// TIA Portal V20 export
FUNCTION_BLOCK "CallEquipment"   // FB29, LAD
TITLE = CallEquipment
AUTHOR : ERsystem_FA2_DH. Kim
// This block contains the logic and futher calls (e.g. sequences, control modules, diagnostics etc.) of the equipment module.
// stored: IsIECCheckEnabled true, MemoryReserve 100, Namespace Unit1.Em5, SetENOAutomatically false
   VAR_INPUT
      ZoneOperationEnable { ExternalWritable := 'False'} : "LWONIK_typeSafetyZoneManualOperation";
   END_VAR
   VAR_IN_OUT
      unitStatus : "LAF_typeUnitStatus";   // Current unit status o be used in this EM
      unitAlarmDB : "LAF_typeAlarms";   // Summarized EM Alarms for the Unit
      emFeedback : "LUC_typeEmFeedback";   // Feedback of the EM to the Unit
   END_VAR
   VAR
      InstSequenceMainPnP { S7_SetPoint := 'True'} : "Unit1.Em5.Sequence_1_MainPnP";   // EM Sequence Instance
      InstSequenceAlignTable { S7_SetPoint := 'True'} : "Unit1.Em5.Sequence_2_AlignTable";
      InstSequenceNgPnP { S7_SetPoint := 'True'} : "Unit1.Em5.Sequence_3_NgPnP";
      InstSequenceGaugeRnR : "Unit1.Em5.Sequence_10_GaugeRnR";
      instMainPnPHomeJob10 : "LAF_SelectJob";
      instMainPnPHomeJob1 : "LAF_SelectJob";
      instMainPnPLoadJob2 : "LAF_SelectJob";
      instMainPnPUnloadJob3 : "LAF_SelectJob";
      instMainPnPAvoidJob4 : "LAF_SelectJob";
      instMainPnPOneLoadJob5 : "LAF_SelectJob";
      instMainPnPOneUnLoadJob6 : "LAF_SelectJob";
      instAlignTableHomeJob1 : "LAF_SelectJob";
      instAlignTableLoadJob2 : "LAF_SelectJob";
      instAlignTableVisionJob3 : "LAF_SelectJob";
      instAlignTableUnloadJob4 : "LAF_SelectJob";
      instAlignTableMotionJob22 : "LAF_SelectJob";
      instNgPnPHomeJob1 : "LAF_SelectJob";
      instNgPnPLoadJob2 : "LAF_SelectJob";
      instNgPnPUnloadJob3 : "LAF_SelectJob";
      instGaugeRnRCommonReadyJob1 : "LAF_SelectJob";
      instGaugeRnRCommonGetMasterPieceJob2 : "LAF_SelectJob";
      instGaugeRnRCommonMainPnPMoveAlignTableStackTableJob3 : "LAF_SelectJob";
      instGaugeRnRCommonMainPnp1ToAlignTableJob4 : "LAF_SelectJob";
      instGaugeRnRCommonMainPnPMoveReelCutConvyorAlignTableJob5 : "LAF_SelectJob";
      instGaugeRnRCommonAlignTableVisionAdjustJob6 : "LAF_SelectJob";
      instGaugeRnR1AlignAlignTableToMainPnP1Job10 { S7_SetPoint := 'True'} : "LAF_SelectJob";
      instGaugeRnR1AlignMainPnPMoveReelCutConvyorAlignTableJob11 { S7_SetPoint := 'True'} : "LAF_SelectJob";
      instGaugeRnR1AlignAlignTableMoveWaitJob12 { S7_SetPoint := 'True'} : "LAF_SelectJob";
      instGaugeRnR1AlignUnloadMasterPieceJob13 { S7_SetPoint := 'True'} : "LAF_SelectJob";
      instGaugeRnR1StackMainPnPMoveReelCutConvyorAlignTableJob15 { S7_SetPoint := 'True'} : "LAF_SelectJob";
      instGaugeRnR1StackAlignTableToMainPnP2Job16 { S7_SetPoint := 'True'} : "LAF_SelectJob";
      instGaugeRnR1StackMainPnPMoveAlignTableJob17 { S7_SetPoint := 'True'} : "LAF_SelectJob";
      instGaugeRnR1StackAlignTableMoveWaitJob18 { S7_SetPoint := 'True'} : "LAF_SelectJob";
      instGaugeRnR1StackMainPnP2ToStackTableJob19 { S7_SetPoint := 'True'} : "LAF_SelectJob";
      instGaugeRnR1StackStackTableToMainPnP2Job20 { S7_SetPoint := 'True'} : "LAF_SelectJob";
      instGaugeRnR1StackMainPnPMoveReelCutConvyorAlignTableJob21 { S7_SetPoint := 'True'} : "LAF_SelectJob";
      instGaugeRnR1StackMainPnP2ToAlignTableJob22 { S7_SetPoint := 'True'} : "LAF_SelectJob";
      instGaugeRnR1StackMainPnPMoveAlignTableJob23 { S7_SetPoint := 'True'} : "LAF_SelectJob";
      instGaugeRnR1StackAlignTableToMainPnP1Job24 { S7_SetPoint := 'True'} : "LAF_SelectJob";
      instGaugeRnR1StackMainPnPMoveReelCutConvyorAlignTableJob25 { S7_SetPoint := 'True'} : "LAF_SelectJob";
      instGaugeRnR1StackUnloadMasterPieceJob26 { S7_SetPoint := 'True'} : "LAF_SelectJob";
      instGaugeRnR3AlignMainPnPMoveReelCutConvyorAlignTableJob30 { S7_SetPoint := 'True'} : "LAF_SelectJob";
      instGaugeRnR3AlignNGPnPLoadMasterPieceJob31 { S7_SetPoint := 'True'} : "LAF_SelectJob";
      instGaugeRnR3AlignMainPnP2MoveAlignTableJob32 { S7_SetPoint := 'True'} : "LAF_SelectJob";
      instGaugeRnR3AlignAlignTableMoveWaitJob33 { S7_SetPoint := 'True'} : "LAF_SelectJob";
      instGaugeRnRCommonCheckCompleteJob39 { S7_SetPoint := 'True'} : "LAF_SelectJob";
      instCmPnp1stCathodeDetectSensor { S7_SetPoint := 'True'} : "LBC_DigitalSignalCn";
      instCmPnp2ndCathodeDetectSensor { S7_SetPoint := 'True'} : "LBC_DigitalSignalCn";
      instCmCathodeAlignTableElectrodeDetectSensor { S7_SetPoint := 'True'} : "LBC_DigitalSignalCn";
      instCmCathodeNgBoxFullSensorDetectSensor { S7_SetPoint := 'True'} : "LBC_DigitalSignalCn";
      instCmCathodeNgBoxDetectSensor { S7_SetPoint := 'True'} : "LBC_DigitalSignalCn";
      instCmCathodeMainPnP1AxisX { S7_SetPoint := 'True'} : "LBC_Axis64Pos_TecPlcCn";
      instCmCathodeMainPnP2AxisX { S7_SetPoint := 'True'} : "LBC_Axis64Pos_TecPlcCn";
      instCmCathodeMainPnP1AxisY { S7_SetPoint := 'True'} : "LBC_Axis64Pos_TecPlcCn";
      instCmCathodeMainPnP1AxisZ { S7_SetPoint := 'True'} : "LBC_Axis64Pos_TecPlcCn";
      instCmCathodeMainPnP2AxisZ { S7_SetPoint := 'True'} : "LBC_Axis64Pos_TecPlcCn";
      instCmCathodeAlignTableAxisX { S7_SetPoint := 'True'} : "LBC_Axis64Pos_TecPlcCn";
      instCmCathodeAlignTableAxisY1 { S7_SetPoint := 'True'} : "LBC_Axis64Pos_TecPlcCn";
      instCmCathodeAlignTableAxisY2 { S7_SetPoint := 'True'} : "LBC_Axis64Pos_TecPlcCn";
      instInterlockCathodeMainPnP1AxisX { S7_SetPoint := 'True'} : "LER_Axis64Pos_InterlockSummary";
      instInterlockCathodeMainPnP1AxisY { S7_SetPoint := 'True'} : "LER_Axis64Pos_InterlockSummary";
      instInterlockCathodeMainPnP1AxisZ { S7_SetPoint := 'True'} : "LER_Axis64Pos_InterlockSummary";
      instInterlockCathodeMainPnP2AxisX { S7_SetPoint := 'True'} : "LER_Axis64Pos_InterlockSummary";
      instInterlockCathodeMainPnP2AxisZ { S7_SetPoint := 'True'} : "LER_Axis64Pos_InterlockSummary";
      instInterlockCathodeAlignTableAxisX { S7_SetPoint := 'True'} : "LER_Axis64Pos_InterlockSummary";
      instInterlockCathodeAlignTableAxisY1 { S7_SetPoint := 'True'} : "LER_Axis64Pos_InterlockSummary";
      instInterlockCathodeAlignTableAxisY2 { S7_SetPoint := 'True'} : "LER_Axis64Pos_InterlockSummary";
      instCathodeMainPnP1AxisXSoftCam : "LER_SoftCam_Interface";
      instCathodeMainPnP2AxisXSoftCam { S7_SetPoint := 'True'} : "LER_SoftCam_Interface";
      instCathodeMainPnP1AxisYSoftCam { S7_SetPoint := 'True'} : "LER_SoftCam_Interface";
      instCathodeMainPnP1AxisZSoftCam { S7_SetPoint := 'True'} : "LER_SoftCam_Interface";
      instCathodeMainPnP2AxisZSoftCam { S7_SetPoint := 'True'} : "LER_SoftCam_Interface";
      instCathodeAlignTableAxisXSoftCam { S7_SetPoint := 'True'} : "LER_SoftCam_Interface";
      instCathodeAlignTableAxisY1SoftCam { S7_SetPoint := 'True'} : "LER_SoftCam_Interface";
      instCathodeAlignTableAxisY2SoftCam { S7_SetPoint := 'True'} : "LER_SoftCam_Interface";
      instCmCathodeMainPnP1RotaryCwCcw { ExternalAccessible := 'False'; ExternalVisible := 'False'; ExternalWritable := 'False'} : "LBC_TwoWayActuatorCn";
      instCmCathodeMainPnP1stSuctionPlateVacuum { ExternalAccessible := 'False'; ExternalVisible := 'False'; ExternalWritable := 'False'} : "LBC_TwoWayActuatorCn";
      instCmCathodeMainPnP2ndSuctionPlateVacuum { ExternalAccessible := 'False'; ExternalVisible := 'False'; ExternalWritable := 'False'} : "LBC_TwoWayActuatorCn";
      instCmCathodeAlignTableSuctionPlateVacuum { ExternalAccessible := 'False'; ExternalVisible := 'False'; ExternalWritable := 'False'; S7_SetPoint := 'True'} : "LBC_TwoWayActuatorCn";
      instCmCathodeGlassCleaning { ExternalAccessible := 'False'; ExternalVisible := 'False'; ExternalWritable := 'False'; S7_SetPoint := 'True'} : "LBC_TwoWayActuatorCn";
      instCmCathodeNgPnpUpDown { ExternalAccessible := 'False'; ExternalVisible := 'False'; ExternalWritable := 'False'; S7_SetPoint := 'True'} : "LBC_TwoWayActuatorCn";
      instCmCathodeNgPnp1stFwdBwd { ExternalAccessible := 'False'; ExternalVisible := 'False'; ExternalWritable := 'False'; S7_SetPoint := 'True'} : "LBC_TwoWayActuatorCn";
      instCmCathodeNgPnp2ndFwdBwd { ExternalAccessible := 'False'; ExternalVisible := 'False'; ExternalWritable := 'False'; S7_SetPoint := 'True'} : "LBC_TwoWayActuatorCn";
      instCmCathodeMaintenanceMovingFixFwdBwd { ExternalAccessible := 'False'; ExternalVisible := 'False'; ExternalWritable := 'False'; S7_SetPoint := 'True'} : "LBC_TwoWayActuatorCn";
      instCmCathodeNgBoxLiftUpDown { ExternalAccessible := 'False'; ExternalVisible := 'False'; ExternalWritable := 'False'; S7_SetPoint := 'True'} : "LBC_TwoWayActuatorCn";
      instCmCathodeNgBoxLockUpDown { ExternalAccessible := 'False'; ExternalVisible := 'False'; ExternalWritable := 'False'; S7_SetPoint := 'True'} : "LBC_TwoWayActuatorCn";
      instCmCathodeNgPnpVaccum { ExternalAccessible := 'False'; ExternalVisible := 'False'; ExternalWritable := 'False'; S7_SetPoint := 'True'} : "LBC_TwoWayActuatorCn";
      instCmCathodeConveyorCoverFwdBwd { S7_SetPoint := 'True'} : "LBC_TwoWayActuatorCn";
      instCmCathodeConveyorPickUpBlower { S7_SetPoint := 'True'} : "LBC_TwoWayActuatorCn";
      instCmCathodeVisionControllerInterface { ExternalAccessible := 'False'; ExternalVisible := 'False'; ExternalWritable := 'False'; S7_SetPoint := 'True'} : "LER_Vision_XGX2000";
      instAlignVisionConversion : "LER_AlignVisionConversion";
      instManageAlarms { ExternalWritable := 'False'} : "LAF_ManageAlarms";
      instEventsPFE : "Unit1.Em5.EventsPFE";
      instLER_BrakeTestCathodeMainPnP1AxisZ : "LER_BrakeTest";
      instLER_BrakeTestCathodeMainPnP2AxisZ { S7_SetPoint := 'True'} : "LER_BrakeTest";
      statUnitStatus { ExternalWritable := 'False'} : "LAF_typeUnitStatus";   // Unit Status used in this EM
      statSlmStatus : Struct
         running { ExternalWritable := 'False'} : Bool;
         powerOff { ExternalWritable := 'False'} : Bool;
      END_STRUCT;
      statAllBrakeTest { ExternalWritable := 'False'} : "LER_typeBrakeTestUnitCommands";
      statTonTime { ExternalAccessible := 'False'; ExternalVisible := 'False'; ExternalWritable := 'False'} : Array[0..1999] of TON_TIME;
      statTofTime { ExternalAccessible := 'False'; ExternalVisible := 'False'; ExternalWritable := 'False'} : Array[0..99] of TOF_TIME;
      statPulse { ExternalAccessible := 'False'; ExternalVisible := 'False'; ExternalWritable := 'False'} : Struct
         miscellaneous : Array[0..99] of Bool;
         workingDone : Struct
            mainPnP : Array[0..99] of Bool;
            alignTable : Array[0..99] of Bool;
            ngPnP : Array[0..99] of Bool;
         END_STRUCT;
         axisEnable : Array[0..99] of Bool;
         brakeTest : Array[0..99] of Bool;
      END_STRUCT;
      statEnableManualCmds : Bool;
      Scan_on : Bool;
      "*** Interlock Axis ***" { ExternalAccessible := 'False'; ExternalVisible := 'False'; ExternalWritable := 'False'} : Bool;
      "cathodeMainPnP1AxisX Home" { S7_SetPoint := 'True'} : "Homing.LER_Axis";
      "cathodeMainPnP1AxisX Jog_CW" { S7_SetPoint := 'True'} : "Jog.LER_Axis";
      "cathodeMainPnP1AxisX Jog_CCW" { S7_SetPoint := 'True'} : "Jog.LER_Axis";
      "cathodeMainPnP1AxisX Position_" { S7_SetPoint := 'True'} : Array[0..5] of "Position.LER_Axis";
      "cathodeMainPnP2AxisX Home" { S7_SetPoint := 'True'} : "Homing.LER_Axis";
      "cathodeMainPnP2AxisX Jog_CW" { S7_SetPoint := 'True'} : "Jog.LER_Axis";
      "cathodeMainPnP2AxisX Jog_CCW" { S7_SetPoint := 'True'} : "Jog.LER_Axis";
      "cathodeMainPnP2AxisX Position_" { S7_SetPoint := 'True'} : Array[0..5] of "Position.LER_Axis";
      "cathodeMainPnP1AxisY Home" { S7_SetPoint := 'True'} : "Homing.LER_Axis";
      "cathodeMainPnP1AxisY Jog_CW" { S7_SetPoint := 'True'} : "Jog.LER_Axis";
      "cathodeMainPnP1AxisY Jog_CCW" { S7_SetPoint := 'True'} : "Jog.LER_Axis";
      "cathodeMainPnP1AxisY Position_" { S7_SetPoint := 'True'} : Array[0..5] of "Position.LER_Axis";
      "cathodeMainPnP1AxisZ Home" { S7_SetPoint := 'True'} : "Homing.LER_Axis";
      "cathodeMainPnP1AxisZ Jog_CW" { S7_SetPoint := 'True'} : "Jog.LER_Axis";
      "cathodeMainPnP1AxisZ Jog_CCW" { S7_SetPoint := 'True'} : "Jog.LER_Axis";
      "cathodeMainPnP1AxisZ Position_" { S7_SetPoint := 'True'} : Array[0..5] of "Position.LER_Axis";
      "cathodeMainPnP2AxisZ Home" { S7_SetPoint := 'True'} : "Homing.LER_Axis";
      "cathodeMainPnP2AxisZ Jog_CW" { S7_SetPoint := 'True'} : "Jog.LER_Axis";
      "cathodeMainPnP2AxisZ Jog_CCW" { S7_SetPoint := 'True'} : "Jog.LER_Axis";
      "cathodeMainPnP2AxisZ Position_" { S7_SetPoint := 'True'} : Array[0..5] of "Position.LER_Axis";
      "cathodeAlignTableAxisX Home" { S7_SetPoint := 'True'} : "Homing.LER_Axis";
      "cathodeAlignTableAxisX Jog_CW" { S7_SetPoint := 'True'} : "Jog.LER_Axis";
      "cathodeAlignTableAxisX Jog_CCW" { S7_SetPoint := 'True'} : "Jog.LER_Axis";
      "cathodeAlignTableAxisX Position_" { S7_SetPoint := 'True'} : Array[0..5] of "Position.LER_Axis";
      "cathodeAlignTableAxisY1 Home" { S7_SetPoint := 'True'} : "Homing.LER_Axis";
      "cathodeAlignTableAxisY1 Jog_CW" { S7_SetPoint := 'True'} : "Jog.LER_Axis";
      "cathodeAlignTableAxisY1 Jog_CCW" { S7_SetPoint := 'True'} : "Jog.LER_Axis";
      "cathodeAlignTableAxisY1 Position_" { S7_SetPoint := 'True'} : Array[0..5] of "Position.LER_Axis";
      "cathodeAlignTableAxisY2 Home" { S7_SetPoint := 'True'} : "Homing.LER_Axis";
      "cathodeAlignTableAxisY2 Jog_CW" { S7_SetPoint := 'True'} : "Jog.LER_Axis";
      "cathodeAlignTableAxisY2 Jog_CCW" { S7_SetPoint := 'True'} : "Jog.LER_Axis";
      "cathodeAlignTableAxisY2 Position_" { S7_SetPoint := 'True'} : Array[0..5] of "Position.LER_Axis";
      "*** Interlock Actuator ******" { ExternalAccessible := 'False'; ExternalVisible := 'False'; ExternalWritable := 'False'} : Bool;
      "cathodeNgBoxLiftUpDown Home" { S7_SetPoint := 'True'} : "Cylinder.LER_Actuator";
      "cathodeNgBoxLiftUpDown Work" { S7_SetPoint := 'True'} : "Cylinder.LER_Actuator";
      "cathodeNgBoxLockUpDown Home" { S7_SetPoint := 'True'} : "Cylinder.LER_Actuator";
      "cathodeNgBoxLockUpDown Work" { S7_SetPoint := 'True'} : "Cylinder.LER_Actuator";
      "cathodeMaintenanceMovingFixFrontFwdBwd Home" { S7_SetPoint := 'True'} : "Cylinder.LER_Actuator";
      "cathodeMaintenanceMovingFixFrontFwdBwd Work" { S7_SetPoint := 'True'} : "Cylinder.LER_Actuator";
      "cathodeGlassCleaning Home" { S7_SetPoint := 'True'} : "Cylinder.LER_Actuator";
      "cathodeGlassCleaning Work" { S7_SetPoint := 'True'} : "Cylinder.LER_Actuator";
      "cathodeNgPnp1stFwdBwd Home" { S7_SetPoint := 'True'} : "Cylinder.LER_Actuator";
      "cathodeNgPnp1stFwdBwd Work" { S7_SetPoint := 'True'} : "Cylinder.LER_Actuator";
      "cathodeNgPnpUpDown Home" { S7_SetPoint := 'True'} : "Cylinder.LER_Actuator";
      "cathodeNgPnpUpDown Work" { S7_SetPoint := 'True'} : "Cylinder.LER_Actuator";
      "cathodeMainPnP1RotaryCwCcw Home" { S7_SetPoint := 'True'} : "Cylinder.LER_Actuator";
      "cathodeMainPnP1RotaryCwCcw Work" { S7_SetPoint := 'True'} : "Cylinder.LER_Actuator";
      "cathodeNgPnp2ndFwdBwd Home" { S7_SetPoint := 'True'} : "Cylinder.LER_Actuator";
      "cathodeNgPnp2ndFwdBwd Work" { S7_SetPoint := 'True'} : "Cylinder.LER_Actuator";
      Tracking_05 { S7_SetPoint := 'True'} : "Unit1.Em5.PartData";
      AXIS7 : "LER_CM_Name";
      AXIS13 : "LER_CM_Name";
      AXIS18 : "LER_CM_Name";
      Cylinder23 : "LER_CM_Name";
      Cylinder28 : "LER_CM_Name";
      Vaccum15 : "LER_CM_Name";
      instAlignVisionHistory { S7_SetPoint := 'True'} : "LER_visionHistory";
      instAlignMoveCalibration { S7_SetPoint := 'True'} : "LER_AlignMoveCalibration";
      instAlignThetaCalibration { S7_SetPoint := 'True'} : "LER_AlignThetaCalibration";
      instAlignSyncMove { S7_SetPoint := 'True'} : "LER_AlignSyncMove";
      citi_Ptrig : Array[0..20] of Bool;
      citiTon : Array[0..20] of TON_TIME;
      citi : Time;
      citiTest : Array[0..20] of Bool;
   END_VAR
   VAR_TEMP
      tempIndex : Int;
      tempScInProduction : Bool;   // Mode Production and StateComplete
      tempScNoProduction : Bool;   // Mode Manual and StateComplete
   END_VAR
   VAR CONSTANT
      delayTime : Time := T#3s;
      TRUE : Bool := TRUE;
      FALSE : Bool := FALSE;
      NO_JOB : DInt;   // No job
      MIN_POSITION_NUMBER : SInt;
      INIT_POSITION_NUMBER : SInt := -1;
   END_VAR
   // // statPulse.brakeTest[0] : Unit Mode Production Rising Edge
   // // statPulse.brakeTest[1] : Unit Mode Production Rising Edge Old
   // // statPulse.brakeTest[10] : Cathode Main PnP 1 Z Axis Error Pulse
   // // statPulse.brakeTest[11] : Cathode Main PnP 2 Z Axis Error Pulse
   VAR_TEMP   // added for the SCL form of the ladder/FBD networks
      _w1 : Bool;
      _w2 : Bool;
      _w3 : Bool;
      _w4 : Bool;
      _w5 : Bool;
      _w6 : Bool;
      _w7 : Bool;
      _w8 : Bool;
      _w9 : Bool;
      _w10 : Bool;
      _w11 : Bool;
   END_VAR
BEGIN

REGION Network 1: BLOCK INFO HEADER
   // (company) / (C) Copyright (year)
   // ---------------------------------------------------------------------------------
   // Title:                             (Title of this block)
   // Comment/Function: (that is implemented in the block)
   // Library/Family:           (that the source is dedicated to)
   // Author:                        (department / person in charge / contact)
   // Target System:          (test system with FW version)
   // Engineering:              TIA Portal (SW version)
   // Restrictions:               (OB types, etc.)
   // Requirements:           (hardware, technological package, etc.)
   // ---------------------------------------------------------------------------------
   // Change log table:
   // Version          | Date             | Signature      | Expert in charge  | Changes applied ------------------------|----------------------|-------------------------|--------------------------------|-----------------------
   // 001.000.000 | yyyy-mm-dd | 0x00000000 | (name of expert) | First released version
END_REGION

REGION Network 2: DESCRIPTION
   // This is a template block provided by the Automation Framework. It can be used to create an own project.
   // The Block Info Header is prepared to put in your own data.
   // Description of the block could be added here and the docu created by Code2Docu.
END_REGION

REGION Network 3: ******************** Unit Input ********************
END_REGION

REGION Network 4: Em6 Relations SoftCam
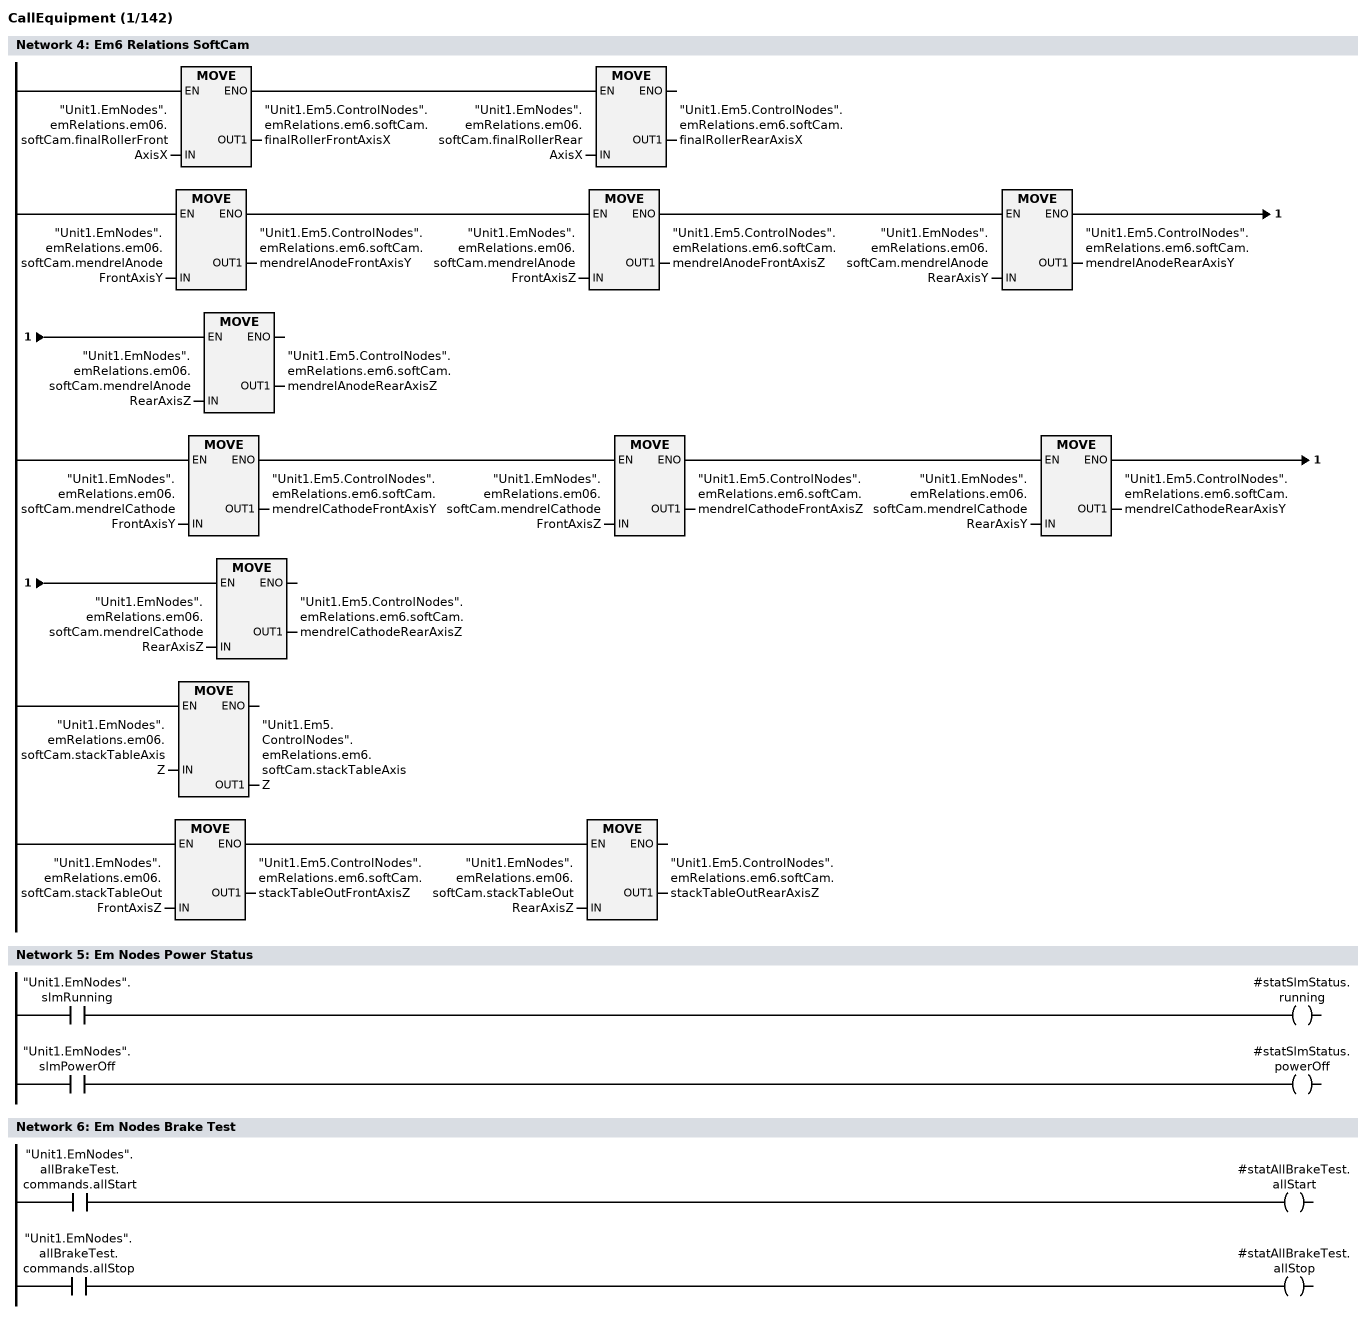
   RUNG wire#powerrail
      Move(in := "Unit1.EmNodes".emRelations.em06.softCam.finalRollerFrontAxisX, out1 => "Unit1.Em5.ControlNodes".emRelations.em6.softCam.finalRollerFrontAxisX)
      Move(in := "Unit1.EmNodes".emRelations.em06.softCam.finalRollerRearAxisX, out1 => "Unit1.Em5.ControlNodes".emRelations.em6.softCam.finalRollerRearAxisX)
   END_RUNG
   RUNG wire#powerrail
      Move(in := "Unit1.EmNodes".emRelations.em06.softCam.mendrelAnodeFrontAxisY, out1 => "Unit1.Em5.ControlNodes".emRelations.em6.softCam.mendrelAnodeFrontAxisY)
      Move(in := "Unit1.EmNodes".emRelations.em06.softCam.mendrelAnodeFrontAxisZ, out1 => "Unit1.Em5.ControlNodes".emRelations.em6.softCam.mendrelAnodeFrontAxisZ)
      Move(in := "Unit1.EmNodes".emRelations.em06.softCam.mendrelAnodeRearAxisY, out1 => "Unit1.Em5.ControlNodes".emRelations.em6.softCam.mendrelAnodeRearAxisY)
      Move(in := "Unit1.EmNodes".emRelations.em06.softCam.mendrelAnodeRearAxisZ, out1 => "Unit1.Em5.ControlNodes".emRelations.em6.softCam.mendrelAnodeRearAxisZ)
   END_RUNG
   RUNG wire#powerrail
      Move(in := "Unit1.EmNodes".emRelations.em06.softCam.mendrelCathodeFrontAxisY, out1 => "Unit1.Em5.ControlNodes".emRelations.em6.softCam.mendrelCathodeFrontAxisY)
      Move(in := "Unit1.EmNodes".emRelations.em06.softCam.mendrelCathodeFrontAxisZ, out1 => "Unit1.Em5.ControlNodes".emRelations.em6.softCam.mendrelCathodeFrontAxisZ)
      Move(in := "Unit1.EmNodes".emRelations.em06.softCam.mendrelCathodeRearAxisY, out1 => "Unit1.Em5.ControlNodes".emRelations.em6.softCam.mendrelCathodeRearAxisY)
      Move(in := "Unit1.EmNodes".emRelations.em06.softCam.mendrelCathodeRearAxisZ, out1 => "Unit1.Em5.ControlNodes".emRelations.em6.softCam.mendrelCathodeRearAxisZ)
   END_RUNG
   RUNG wire#powerrail
      Move(in := "Unit1.EmNodes".emRelations.em06.softCam.stackTableAxisZ, out1 => "Unit1.Em5.ControlNodes".emRelations.em6.softCam.stackTableAxisZ)
   END_RUNG
   RUNG wire#powerrail
      Move(in := "Unit1.EmNodes".emRelations.em06.softCam.stackTableOutFrontAxisZ, out1 => "Unit1.Em5.ControlNodes".emRelations.em6.softCam.stackTableOutFrontAxisZ)
      Move(in := "Unit1.EmNodes".emRelations.em06.softCam.stackTableOutRearAxisZ, out1 => "Unit1.Em5.ControlNodes".emRelations.em6.softCam.stackTableOutRearAxisZ)
   END_RUNG
   // the same network as SCL:
   "Unit1.Em5.ControlNodes".emRelations.em6.softCam.finalRollerFrontAxisX := "Unit1.EmNodes".emRelations.em06.softCam.finalRollerFrontAxisX;
   "Unit1.Em5.ControlNodes".emRelations.em6.softCam.finalRollerRearAxisX := "Unit1.EmNodes".emRelations.em06.softCam.finalRollerRearAxisX;
   "Unit1.Em5.ControlNodes".emRelations.em6.softCam.mendrelAnodeFrontAxisY := "Unit1.EmNodes".emRelations.em06.softCam.mendrelAnodeFrontAxisY;
   "Unit1.Em5.ControlNodes".emRelations.em6.softCam.mendrelAnodeFrontAxisZ := "Unit1.EmNodes".emRelations.em06.softCam.mendrelAnodeFrontAxisZ;
   "Unit1.Em5.ControlNodes".emRelations.em6.softCam.mendrelAnodeRearAxisY := "Unit1.EmNodes".emRelations.em06.softCam.mendrelAnodeRearAxisY;
   "Unit1.Em5.ControlNodes".emRelations.em6.softCam.mendrelAnodeRearAxisZ := "Unit1.EmNodes".emRelations.em06.softCam.mendrelAnodeRearAxisZ;
   "Unit1.Em5.ControlNodes".emRelations.em6.softCam.mendrelCathodeFrontAxisY := "Unit1.EmNodes".emRelations.em06.softCam.mendrelCathodeFrontAxisY;
   "Unit1.Em5.ControlNodes".emRelations.em6.softCam.mendrelCathodeFrontAxisZ := "Unit1.EmNodes".emRelations.em06.softCam.mendrelCathodeFrontAxisZ;
   "Unit1.Em5.ControlNodes".emRelations.em6.softCam.mendrelCathodeRearAxisY := "Unit1.EmNodes".emRelations.em06.softCam.mendrelCathodeRearAxisY;
   "Unit1.Em5.ControlNodes".emRelations.em6.softCam.mendrelCathodeRearAxisZ := "Unit1.EmNodes".emRelations.em06.softCam.mendrelCathodeRearAxisZ;
   "Unit1.Em5.ControlNodes".emRelations.em6.softCam.stackTableAxisZ := "Unit1.EmNodes".emRelations.em06.softCam.stackTableAxisZ;
   "Unit1.Em5.ControlNodes".emRelations.em6.softCam.stackTableOutFrontAxisZ := "Unit1.EmNodes".emRelations.em06.softCam.stackTableOutFrontAxisZ;
   "Unit1.Em5.ControlNodes".emRelations.em6.softCam.stackTableOutRearAxisZ := "Unit1.EmNodes".emRelations.em06.softCam.stackTableOutRearAxisZ;
END_REGION

REGION Network 5: Em Nodes Power Status
   RUNG wire#powerrail
      Contact( "Unit1.EmNodes".slmRunning )
      Coil( #statSlmStatus.running )
   END_RUNG
   RUNG wire#powerrail
      Contact( "Unit1.EmNodes".slmPowerOff )
      Coil( #statSlmStatus.powerOff )
   END_RUNG
   // the same network as SCL:
   #statSlmStatus.running := "Unit1.EmNodes".slmRunning;
   #statSlmStatus.powerOff := "Unit1.EmNodes".slmPowerOff;
END_REGION

REGION Network 6: Em Nodes Brake Test
   RUNG wire#powerrail
      Contact( "Unit1.EmNodes".allBrakeTest.commands.allStart )
      Coil( #statAllBrakeTest.allStart )
   END_RUNG
   RUNG wire#powerrail
      Contact( "Unit1.EmNodes".allBrakeTest.commands.allStop )
      Coil( #statAllBrakeTest.allStop )
   END_RUNG
   // the same network as SCL:
   #statAllBrakeTest.allStart := "Unit1.EmNodes".allBrakeTest.commands.allStart;
   #statAllBrakeTest.allStop := "Unit1.EmNodes".allBrakeTest.commands.allStop;
END_REGION

REGION Network 7: *************** Equipment Control **************************
END_REGION

REGION Network 8: Interlink EM to Unit
   // This block links and unlinks the EM from the unit. The command to link/unlink can be set directly by the inputs of the block (e.g. to link/unlink based on any program logic) or through the InOut "hmiInterface". The block changes the output "isLinked" to true/false, depending on the command and if a change is allowed. A changed is allowed if the unit is in state aborted, clearing or stopped. The output "isLinked" is send back to the unit. If the EM is not linked, the unit ignores this EM.
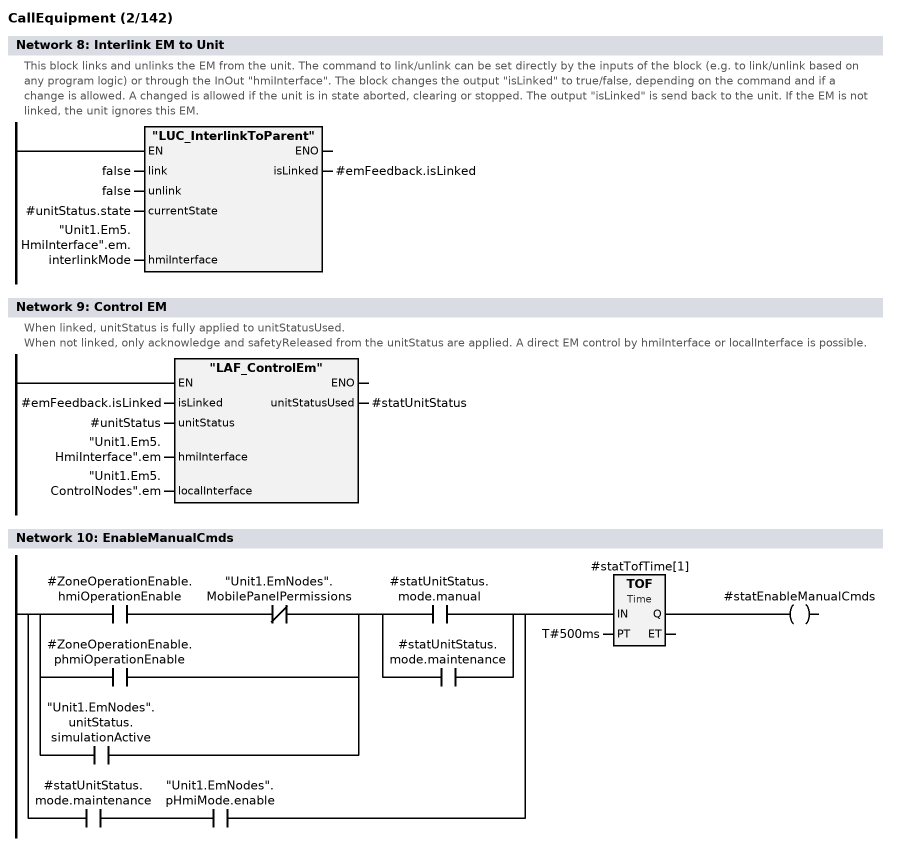
   RUNG wire#powerrail
      "LUC_InterlinkToParent"(link := false, unlink := false, currentState := #unitStatus.state, hmiInterface := "Unit1.Em5.HmiInterface".em.interlinkMode, isLinked => #emFeedback.isLinked)
   END_RUNG
   // the same network as SCL:
   "LUC_InterlinkToParent"(link := false,
                           unlink := false,
                           currentState := #unitStatus.state,
                           hmiInterface := "Unit1.Em5.HmiInterface".em.interlinkMode,
                           isLinked => #emFeedback.isLinked);
END_REGION

REGION Network 9: Control EM
   // When linked, unitStatus is fully applied to unitStatusUsed.
   // When not linked, only acknowledge and safetyReleased from the unitStatus are applied. A direct EM control by hmiInterface or localInterface is possible.
   RUNG wire#powerrail
      "LAF_ControlEm"(isLinked := #emFeedback.isLinked, unitStatus := #unitStatus, hmiInterface := "Unit1.Em5.HmiInterface".em, localInterface := "Unit1.Em5.ControlNodes".em, unitStatusUsed => #statUnitStatus)
   END_RUNG
   // the same network as SCL:
   "LAF_ControlEm"(isLinked := #emFeedback.isLinked,
                   unitStatus := #unitStatus,
                   hmiInterface := "Unit1.Em5.HmiInterface".em,
                   localInterface := "Unit1.Em5.ControlNodes".em,
                   unitStatusUsed => #statUnitStatus);
END_REGION

REGION Network 10: EnableManualCmds
   RUNG wire#powerrail
      Contact( #ZoneOperationEnable.hmiOperationEnable )
      I_Contact( "Unit1.EmNodes".MobilePanelPermissions )
      wire#w1
      Contact( #statUnitStatus.mode.manual )
      wire#w2
      { S7_Templates := "time_type := Time" } #statTofTime[1].TOF(pt := T#500ms, et =>)
      Coil( #statEnableManualCmds )
   END_RUNG
   RUNG wire#powerrail
      Contact( #ZoneOperationEnable.phmiOperationEnable )
   END_RUNG wire#w1
   RUNG wire#powerrail
      Contact( "Unit1.EmNodes".unitStatus.simulationActive )
   END_RUNG wire#w1
   RUNG wire#w1
      Contact( #statUnitStatus.mode.maintenance )
   END_RUNG wire#w2
   RUNG wire#powerrail
      Contact( #statUnitStatus.mode.maintenance )
      Contact( "Unit1.EmNodes".pHmiMode.enable )
   END_RUNG wire#w2
   // the same network as SCL:
   #statTofTime[1].TOF(IN := (((#ZoneOperationEnable.hmiOperationEnable AND NOT "Unit1.EmNodes".MobilePanelPermissions) OR #ZoneOperationEnable.phmiOperationEnable OR "Unit1.EmNodes".unitStatus.simulationActive) AND (#statUnitStatus.mode.manual OR #statUnitStatus.mode.maintenance)) OR (#statUnitStatus.mode.maintenance AND "Unit1.EmNodes".pHmiMode.enable),
                       PT := T#500ms);
   #statEnableManualCmds := #statTofTime[1].Q;
END_REGION

REGION Network 11: DryRun Config Setting
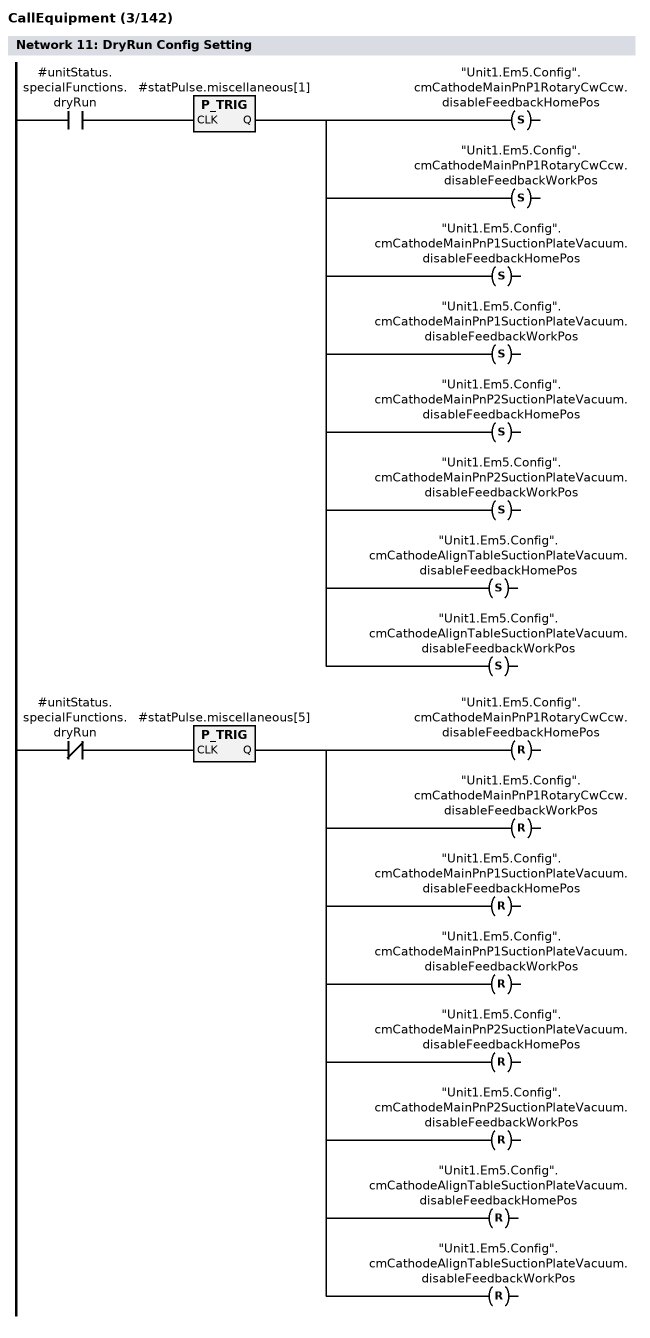
   RUNG wire#powerrail
      Contact( #unitStatus.specialFunctions.dryRun )
      P_Trig( #statPulse.miscellaneous[1] )
      wire#w1
      S_Coil( "Unit1.Em5.Config".cmCathodeMainPnP1RotaryCwCcw.disableFeedbackHomePos )
   END_RUNG
   RUNG wire#w1
      S_Coil( "Unit1.Em5.Config".cmCathodeMainPnP1RotaryCwCcw.disableFeedbackWorkPos )
   END_RUNG
   RUNG wire#w1
      S_Coil( "Unit1.Em5.Config".cmCathodeMainPnP1SuctionPlateVacuum.disableFeedbackHomePos )
   END_RUNG
   RUNG wire#w1
      S_Coil( "Unit1.Em5.Config".cmCathodeMainPnP1SuctionPlateVacuum.disableFeedbackWorkPos )
   END_RUNG
   RUNG wire#w1
      S_Coil( "Unit1.Em5.Config".cmCathodeMainPnP2SuctionPlateVacuum.disableFeedbackHomePos )
   END_RUNG
   RUNG wire#w1
      S_Coil( "Unit1.Em5.Config".cmCathodeMainPnP2SuctionPlateVacuum.disableFeedbackWorkPos )
   END_RUNG
   RUNG wire#w1
      S_Coil( "Unit1.Em5.Config".cmCathodeAlignTableSuctionPlateVacuum.disableFeedbackHomePos )
   END_RUNG
   RUNG wire#w1
      S_Coil( "Unit1.Em5.Config".cmCathodeAlignTableSuctionPlateVacuum.disableFeedbackWorkPos )
   END_RUNG
   RUNG wire#powerrail
      I_Contact( #unitStatus.specialFunctions.dryRun )
      P_Trig( #statPulse.miscellaneous[5] )
      wire#w2
      R_Coil( "Unit1.Em5.Config".cmCathodeMainPnP1RotaryCwCcw.disableFeedbackHomePos )
   END_RUNG
   RUNG wire#w2
      R_Coil( "Unit1.Em5.Config".cmCathodeMainPnP1RotaryCwCcw.disableFeedbackWorkPos )
   END_RUNG
   RUNG wire#w2
      R_Coil( "Unit1.Em5.Config".cmCathodeMainPnP1SuctionPlateVacuum.disableFeedbackHomePos )
   END_RUNG
   RUNG wire#w2
      R_Coil( "Unit1.Em5.Config".cmCathodeMainPnP1SuctionPlateVacuum.disableFeedbackWorkPos )
   END_RUNG
   RUNG wire#w2
      R_Coil( "Unit1.Em5.Config".cmCathodeMainPnP2SuctionPlateVacuum.disableFeedbackHomePos )
   END_RUNG
   RUNG wire#w2
      R_Coil( "Unit1.Em5.Config".cmCathodeMainPnP2SuctionPlateVacuum.disableFeedbackWorkPos )
   END_RUNG
   RUNG wire#w2
      R_Coil( "Unit1.Em5.Config".cmCathodeAlignTableSuctionPlateVacuum.disableFeedbackHomePos )
   END_RUNG
   RUNG wire#w2
      R_Coil( "Unit1.Em5.Config".cmCathodeAlignTableSuctionPlateVacuum.disableFeedbackWorkPos )
   END_RUNG
   // the same network as SCL:
   #_w1 := #unitStatus.specialFunctions.dryRun AND NOT #statPulse.miscellaneous[1];   // rising edge
   #statPulse.miscellaneous[1] := #unitStatus.specialFunctions.dryRun;
   IF #_w1 THEN
       "Unit1.Em5.Config".cmCathodeMainPnP1RotaryCwCcw.disableFeedbackHomePos := TRUE;
       "Unit1.Em5.Config".cmCathodeMainPnP1RotaryCwCcw.disableFeedbackWorkPos := TRUE;
       "Unit1.Em5.Config".cmCathodeMainPnP1SuctionPlateVacuum.disableFeedbackHomePos := TRUE;
       "Unit1.Em5.Config".cmCathodeMainPnP1SuctionPlateVacuum.disableFeedbackWorkPos := TRUE;
       "Unit1.Em5.Config".cmCathodeMainPnP2SuctionPlateVacuum.disableFeedbackHomePos := TRUE;
       "Unit1.Em5.Config".cmCathodeMainPnP2SuctionPlateVacuum.disableFeedbackWorkPos := TRUE;
       "Unit1.Em5.Config".cmCathodeAlignTableSuctionPlateVacuum.disableFeedbackHomePos := TRUE;
       "Unit1.Em5.Config".cmCathodeAlignTableSuctionPlateVacuum.disableFeedbackWorkPos := TRUE;
   END_IF;
   #_w2 := NOT #unitStatus.specialFunctions.dryRun AND NOT #statPulse.miscellaneous[5];   // rising edge
   #statPulse.miscellaneous[5] := NOT #unitStatus.specialFunctions.dryRun;
   IF #_w2 THEN
       "Unit1.Em5.Config".cmCathodeMainPnP1RotaryCwCcw.disableFeedbackHomePos := FALSE;
       "Unit1.Em5.Config".cmCathodeMainPnP1RotaryCwCcw.disableFeedbackWorkPos := FALSE;
       "Unit1.Em5.Config".cmCathodeMainPnP1SuctionPlateVacuum.disableFeedbackHomePos := FALSE;
       "Unit1.Em5.Config".cmCathodeMainPnP1SuctionPlateVacuum.disableFeedbackWorkPos := FALSE;
       "Unit1.Em5.Config".cmCathodeMainPnP2SuctionPlateVacuum.disableFeedbackHomePos := FALSE;
       "Unit1.Em5.Config".cmCathodeMainPnP2SuctionPlateVacuum.disableFeedbackWorkPos := FALSE;
       "Unit1.Em5.Config".cmCathodeAlignTableSuctionPlateVacuum.disableFeedbackHomePos := FALSE;
       "Unit1.Em5.Config".cmCathodeAlignTableSuctionPlateVacuum.disableFeedbackWorkPos := FALSE;
   END_IF;
END_REGION

REGION Network 12: *************** Control Modules (Sensors) ********************
   // Call control modules that are sensors before the em logic (jobs and sequence), so that the latest value is used in the logic.
END_REGION

REGION Network 13: Call Pnp1stCathodeDetectSensor (LBC_DigitalSignal)
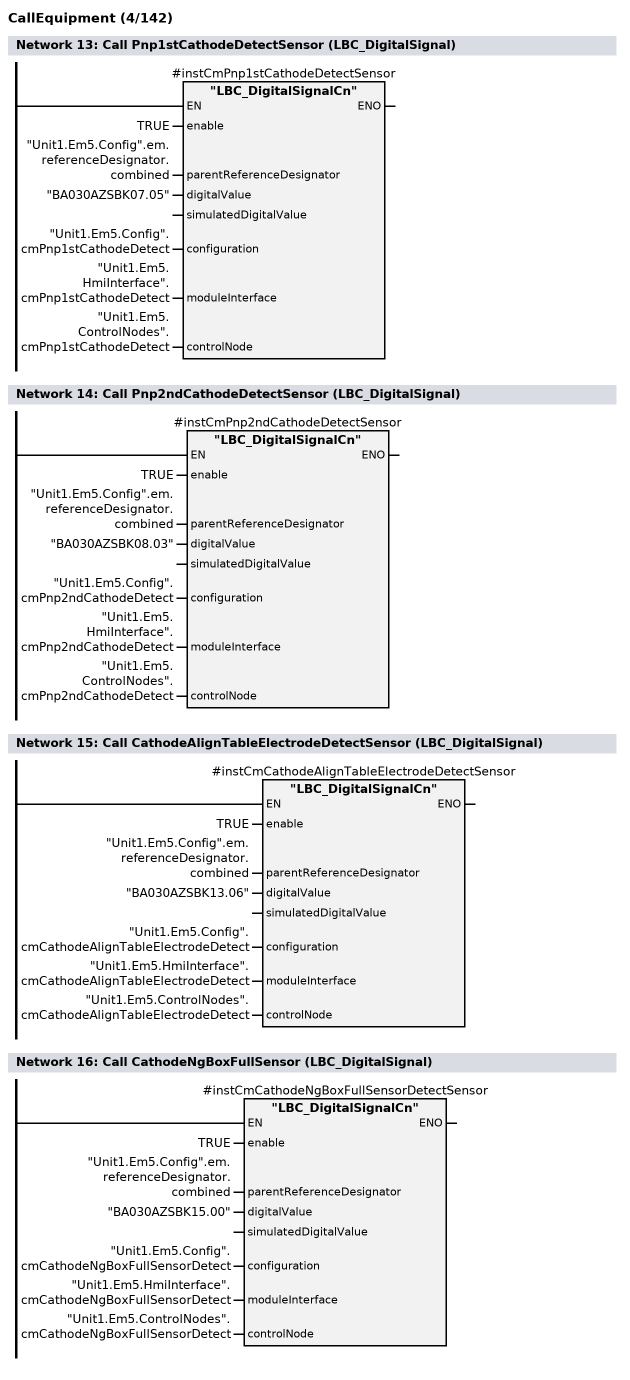
   RUNG wire#powerrail
      #instCmPnp1stCathodeDetectSensor(enable := TRUE, parentReferenceDesignator := "Unit1.Em5.Config".em.referenceDesignator.combined, digitalValue := "BA030AZSBK07.05", simulatedDigitalValue :=, configuration := "Unit1.Em5.Config".cmPnp1stCathodeDetect, moduleInterface := "Unit1.Em5.HmiInterface".cmPnp1stCathodeDetect, controlNode := "Unit1.Em5.ControlNodes".cmPnp1stCathodeDetect)
   END_RUNG
   // the same network as SCL:
   #instCmPnp1stCathodeDetectSensor(enable := TRUE,   // "LBC_DigitalSignalCn"
                           parentReferenceDesignator := "Unit1.Em5.Config".em.referenceDesignator.combined,
                           digitalValue := "BA030AZSBK07.05",
                           configuration := "Unit1.Em5.Config".cmPnp1stCathodeDetect,
                           moduleInterface := "Unit1.Em5.HmiInterface".cmPnp1stCathodeDetect,
                           controlNode := "Unit1.Em5.ControlNodes".cmPnp1stCathodeDetect);
END_REGION

REGION Network 14: Call Pnp2ndCathodeDetectSensor (LBC_DigitalSignal)
   RUNG wire#powerrail
      #instCmPnp2ndCathodeDetectSensor(enable := TRUE, parentReferenceDesignator := "Unit1.Em5.Config".em.referenceDesignator.combined, digitalValue := "BA030AZSBK08.03", simulatedDigitalValue :=, configuration := "Unit1.Em5.Config".cmPnp2ndCathodeDetect, moduleInterface := "Unit1.Em5.HmiInterface".cmPnp2ndCathodeDetect, controlNode := "Unit1.Em5.ControlNodes".cmPnp2ndCathodeDetect)
   END_RUNG
   // the same network as SCL:
   #instCmPnp2ndCathodeDetectSensor(enable := TRUE,   // "LBC_DigitalSignalCn"
                           parentReferenceDesignator := "Unit1.Em5.Config".em.referenceDesignator.combined,
                           digitalValue := "BA030AZSBK08.03",
                           configuration := "Unit1.Em5.Config".cmPnp2ndCathodeDetect,
                           moduleInterface := "Unit1.Em5.HmiInterface".cmPnp2ndCathodeDetect,
                           controlNode := "Unit1.Em5.ControlNodes".cmPnp2ndCathodeDetect);
END_REGION

REGION Network 15: Call CathodeAlignTableElectrodeDetectSensor (LBC_DigitalSignal)
   RUNG wire#powerrail
      #instCmCathodeAlignTableElectrodeDetectSensor(enable := TRUE, parentReferenceDesignator := "Unit1.Em5.Config".em.referenceDesignator.combined, digitalValue := "BA030AZSBK13.06", simulatedDigitalValue :=, configuration := "Unit1.Em5.Config".cmCathodeAlignTableElectrodeDetect, moduleInterface := "Unit1.Em5.HmiInterface".cmCathodeAlignTableElectrodeDetect, controlNode := "Unit1.Em5.ControlNodes".cmCathodeAlignTableElectrodeDetect)
   END_RUNG
   // the same network as SCL:
   #instCmCathodeAlignTableElectrodeDetectSensor(enable := TRUE,   // "LBC_DigitalSignalCn"
                           parentReferenceDesignator := "Unit1.Em5.Config".em.referenceDesignator.combined,
                           digitalValue := "BA030AZSBK13.06",
                           configuration := "Unit1.Em5.Config".cmCathodeAlignTableElectrodeDetect,
                           moduleInterface := "Unit1.Em5.HmiInterface".cmCathodeAlignTableElectrodeDetect,
                           controlNode := "Unit1.Em5.ControlNodes".cmCathodeAlignTableElectrodeDetect);
END_REGION

REGION Network 16: Call CathodeNgBoxFullSensor (LBC_DigitalSignal)
   RUNG wire#powerrail
      #instCmCathodeNgBoxFullSensorDetectSensor(enable := TRUE, parentReferenceDesignator := "Unit1.Em5.Config".em.referenceDesignator.combined, digitalValue := "BA030AZSBK15.00", simulatedDigitalValue :=, configuration := "Unit1.Em5.Config".cmCathodeNgBoxFullSensorDetect, moduleInterface := "Unit1.Em5.HmiInterface".cmCathodeNgBoxFullSensorDetect, controlNode := "Unit1.Em5.ControlNodes".cmCathodeNgBoxFullSensorDetect)
   END_RUNG
   // the same network as SCL:
   #instCmCathodeNgBoxFullSensorDetectSensor(enable := TRUE,   // "LBC_DigitalSignalCn"
                           parentReferenceDesignator := "Unit1.Em5.Config".em.referenceDesignator.combined,
                           digitalValue := "BA030AZSBK15.00",
                           configuration := "Unit1.Em5.Config".cmCathodeNgBoxFullSensorDetect,
                           moduleInterface := "Unit1.Em5.HmiInterface".cmCathodeNgBoxFullSensorDetect,
                           controlNode := "Unit1.Em5.ControlNodes".cmCathodeNgBoxFullSensorDetect);
END_REGION

REGION Network 17: Call CathodeNgBoxDetectSensor (LBC_DigitalSignal)
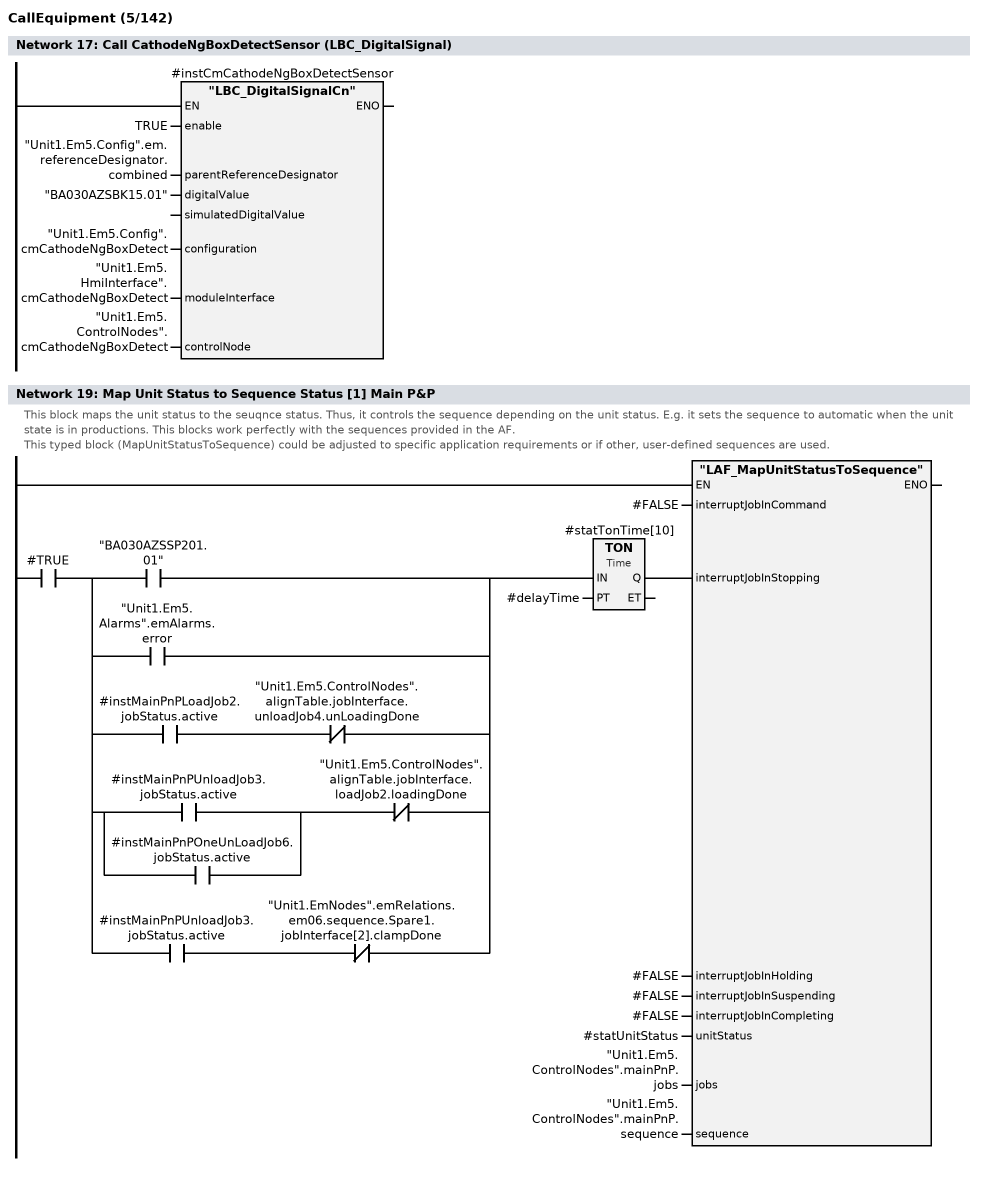
   RUNG wire#powerrail
      #instCmCathodeNgBoxDetectSensor(enable := TRUE, parentReferenceDesignator := "Unit1.Em5.Config".em.referenceDesignator.combined, digitalValue := "BA030AZSBK15.01", simulatedDigitalValue :=, configuration := "Unit1.Em5.Config".cmCathodeNgBoxDetect, moduleInterface := "Unit1.Em5.HmiInterface".cmCathodeNgBoxDetect, controlNode := "Unit1.Em5.ControlNodes".cmCathodeNgBoxDetect)
   END_RUNG
   // the same network as SCL:
   #instCmCathodeNgBoxDetectSensor(enable := TRUE,   // "LBC_DigitalSignalCn"
                           parentReferenceDesignator := "Unit1.Em5.Config".em.referenceDesignator.combined,
                           digitalValue := "BA030AZSBK15.01",
                           configuration := "Unit1.Em5.Config".cmCathodeNgBoxDetect,
                           moduleInterface := "Unit1.Em5.HmiInterface".cmCathodeNgBoxDetect,
                           controlNode := "Unit1.Em5.ControlNodes".cmCathodeNgBoxDetect);
END_REGION

REGION Network 18: *************** Equipment Logic ***************************
END_REGION

REGION Network 19: Map Unit Status to Sequence Status [1] Main P&P
   // This block maps the unit status to the seuqnce status. Thus, it controls the sequence depending on the unit status. E.g. it sets the sequence to automatic when the unit state is in productions. This blocks work perfectly with the sequences provided in the AF. 
   // This typed block (MapUnitStatusToSequence) could be adjusted to specific application requirements or if other, user-defined sequences are used.
   RUNG wire#powerrail
      "LAF_MapUnitStatusToSequence"(interruptJobInStopping := wire#w4, interruptJobInCommand := #FALSE, interruptJobInHolding := #FALSE, interruptJobInSuspending := #FALSE, interruptJobInCompleting := #FALSE, unitStatus := #statUnitStatus, jobs := "Unit1.Em5.ControlNodes".mainPnP.jobs, sequence := "Unit1.Em5.ControlNodes".mainPnP.sequence)
   END_RUNG
   RUNG wire#powerrail
      Contact( #TRUE )
      wire#w1
      Contact( "BA030AZSSP201.01" )
      wire#w2
      { S7_Templates := "time_type := Time" } #statTonTime[10].TON(pt := #delayTime, et =>)
   END_RUNG wire#w4
   RUNG wire#w1
      Contact( "Unit1.Em5.Alarms".emAlarms.error )
   END_RUNG wire#w2
   RUNG wire#w1
      Contact( #instMainPnPLoadJob2.jobStatus.active )
      I_Contact( "Unit1.Em5.ControlNodes".alignTable.jobInterface.unloadJob4.unLoadingDone )
   END_RUNG wire#w2
   RUNG wire#w1
      Contact( #instMainPnPUnloadJob3.jobStatus.active )
      wire#w3
      I_Contact( "Unit1.Em5.ControlNodes".alignTable.jobInterface.loadJob2.loadingDone )
   END_RUNG wire#w2
   RUNG wire#w1
      Contact( #instMainPnPOneUnLoadJob6.jobStatus.active )
   END_RUNG wire#w3
   RUNG wire#w1
      Contact( #instMainPnPUnloadJob3.jobStatus.active )
      I_Contact( "Unit1.EmNodes".emRelations.em06.sequence.Spare1.jobInterface[2].clampDone )
   END_RUNG wire#w2
   // the same network as SCL:
   #statTonTime[10].TON(IN := #TRUE AND ("BA030AZSSP201.01" OR "Unit1.Em5.Alarms".emAlarms.error OR (#instMainPnPLoadJob2.jobStatus.active AND NOT "Unit1.Em5.ControlNodes".alignTable.jobInterface.unloadJob4.unLoadingDone) OR ((#instMainPnPUnloadJob3.jobStatus.active OR #instMainPnPOneUnLoadJob6.jobStatus.active) AND NOT "Unit1.Em5.ControlNodes".alignTable.jobInterface.loadJob2.loadingDone) OR (#instMainPnPUnloadJob3.jobStatus.active AND NOT "Unit1.EmNodes".emRelations.em06.sequence.Spare1.jobInterface[2].clampDone)),
                        PT := #delayTime);
   "LAF_MapUnitStatusToSequence"(interruptJobInCommand := #FALSE,
                           interruptJobInStopping := #statTonTime[10].Q,
                           interruptJobInHolding := #FALSE,
                           interruptJobInSuspending := #FALSE,
                           interruptJobInCompleting := #FALSE,
                           unitStatus := #statUnitStatus,
                           jobs := "Unit1.Em5.ControlNodes".mainPnP.jobs,
                           sequence := "Unit1.Em5.ControlNodes".mainPnP.sequence);
END_REGION

REGION Network 20: Map Unit Status to Sequence Status [2] Align Table
   // This block maps the unit status to the seuqnce status. Thus, it controls the sequence depending on the unit status. E.g. it sets the sequence to automatic when the unit state is in productions. This blocks work perfectly with the sequences provided in the AF. 
   // This typed block (MapUnitStatusToSequence) could be adjusted to specific application requirements or if other, user-defined sequences are used.
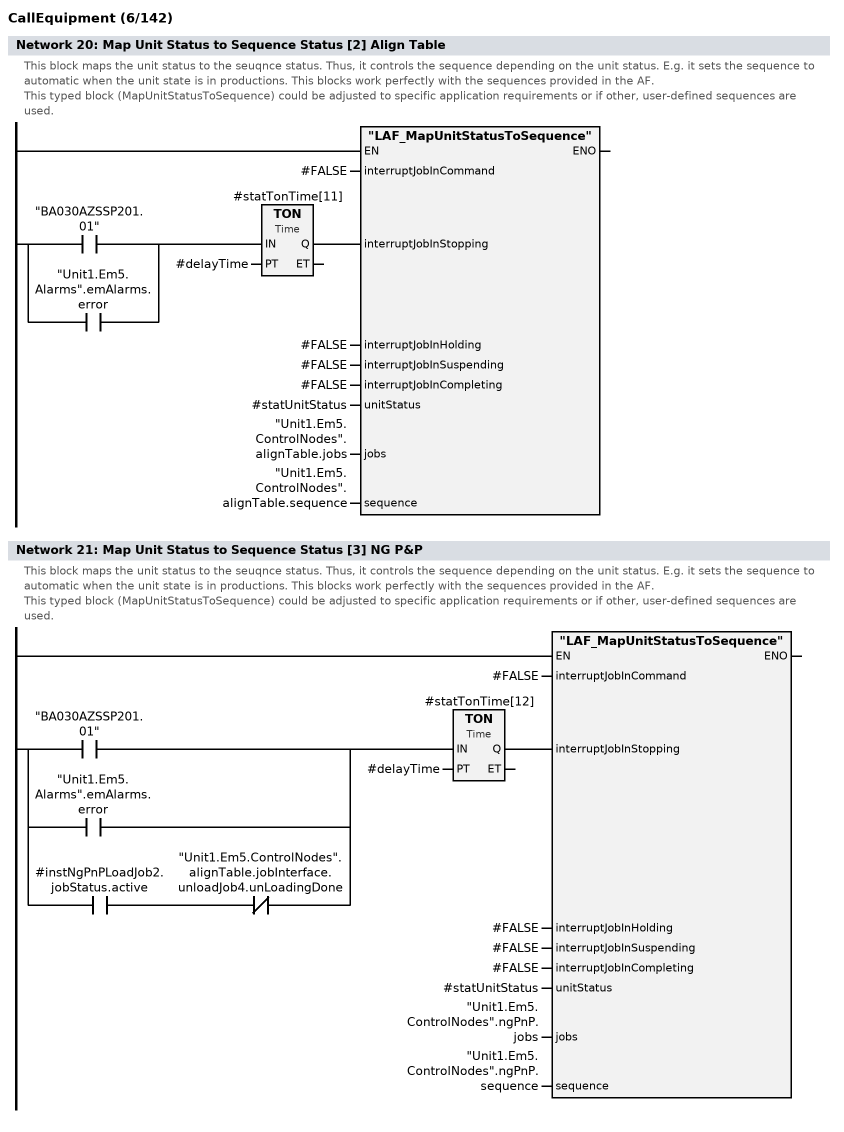
   RUNG wire#powerrail
      "LAF_MapUnitStatusToSequence"(interruptJobInStopping := wire#w2, interruptJobInCommand := #FALSE, interruptJobInHolding := #FALSE, interruptJobInSuspending := #FALSE, interruptJobInCompleting := #FALSE, unitStatus := #statUnitStatus, jobs := "Unit1.Em5.ControlNodes".alignTable.jobs, sequence := "Unit1.Em5.ControlNodes".alignTable.sequence)
   END_RUNG
   RUNG wire#powerrail
      Contact( "BA030AZSSP201.01" )
      wire#w1
      { S7_Templates := "time_type := Time" } #statTonTime[11].TON(pt := #delayTime, et =>)
   END_RUNG wire#w2
   RUNG wire#powerrail
      Contact( "Unit1.Em5.Alarms".emAlarms.error )
   END_RUNG wire#w1
   // the same network as SCL:
   #statTonTime[11].TON(IN := "BA030AZSSP201.01" OR "Unit1.Em5.Alarms".emAlarms.error, PT := #delayTime);
   "LAF_MapUnitStatusToSequence"(interruptJobInCommand := #FALSE,
                           interruptJobInStopping := #statTonTime[11].Q,
                           interruptJobInHolding := #FALSE,
                           interruptJobInSuspending := #FALSE,
                           interruptJobInCompleting := #FALSE,
                           unitStatus := #statUnitStatus,
                           jobs := "Unit1.Em5.ControlNodes".alignTable.jobs,
                           sequence := "Unit1.Em5.ControlNodes".alignTable.sequence);
END_REGION

REGION Network 21: Map Unit Status to Sequence Status [3] NG P&P
   // This block maps the unit status to the seuqnce status. Thus, it controls the sequence depending on the unit status. E.g. it sets the sequence to automatic when the unit state is in productions. This blocks work perfectly with the sequences provided in the AF. 
   // This typed block (MapUnitStatusToSequence) could be adjusted to specific application requirements or if other, user-defined sequences are used.
   RUNG wire#powerrail
      "LAF_MapUnitStatusToSequence"(interruptJobInStopping := wire#w2, interruptJobInCommand := #FALSE, interruptJobInHolding := #FALSE, interruptJobInSuspending := #FALSE, interruptJobInCompleting := #FALSE, unitStatus := #statUnitStatus, jobs := "Unit1.Em5.ControlNodes".ngPnP.jobs, sequence := "Unit1.Em5.ControlNodes".ngPnP.sequence)
   END_RUNG
   RUNG wire#powerrail
      Contact( "BA030AZSSP201.01" )
      wire#w1
      { S7_Templates := "time_type := Time" } #statTonTime[12].TON(pt := #delayTime, et =>)
   END_RUNG wire#w2
   RUNG wire#powerrail
      Contact( "Unit1.Em5.Alarms".emAlarms.error )
   END_RUNG wire#w1
   RUNG wire#powerrail
      Contact( #instNgPnPLoadJob2.jobStatus.active )
      I_Contact( "Unit1.Em5.ControlNodes".alignTable.jobInterface.unloadJob4.unLoadingDone )
   END_RUNG wire#w1
   // the same network as SCL:
   #statTonTime[12].TON(IN := "BA030AZSSP201.01" OR "Unit1.Em5.Alarms".emAlarms.error OR (#instNgPnPLoadJob2.jobStatus.active AND NOT "Unit1.Em5.ControlNodes".alignTable.jobInterface.unloadJob4.unLoadingDone),
                        PT := #delayTime);
   "LAF_MapUnitStatusToSequence"(interruptJobInCommand := #FALSE,
                           interruptJobInStopping := #statTonTime[12].Q,
                           interruptJobInHolding := #FALSE,
                           interruptJobInSuspending := #FALSE,
                           interruptJobInCompleting := #FALSE,
                           unitStatus := #statUnitStatus,
                           jobs := "Unit1.Em5.ControlNodes".ngPnP.jobs,
                           sequence := "Unit1.Em5.ControlNodes".ngPnP.sequence);
END_REGION

REGION Network 22: Map Unit Status to Sequence Status [4] Gague R&R
   // This block maps the unit status to the seuqnce status. Thus, it controls the sequence depending on the unit status. E.g. it sets the sequence to automatic when the unit state is in productions. This blocks work perfectly with the sequences provided in the AF. 
   // This typed block (MapUnitStatusToSequence) could be adjusted to specific application requirements or if other, user-defined sequences are used.
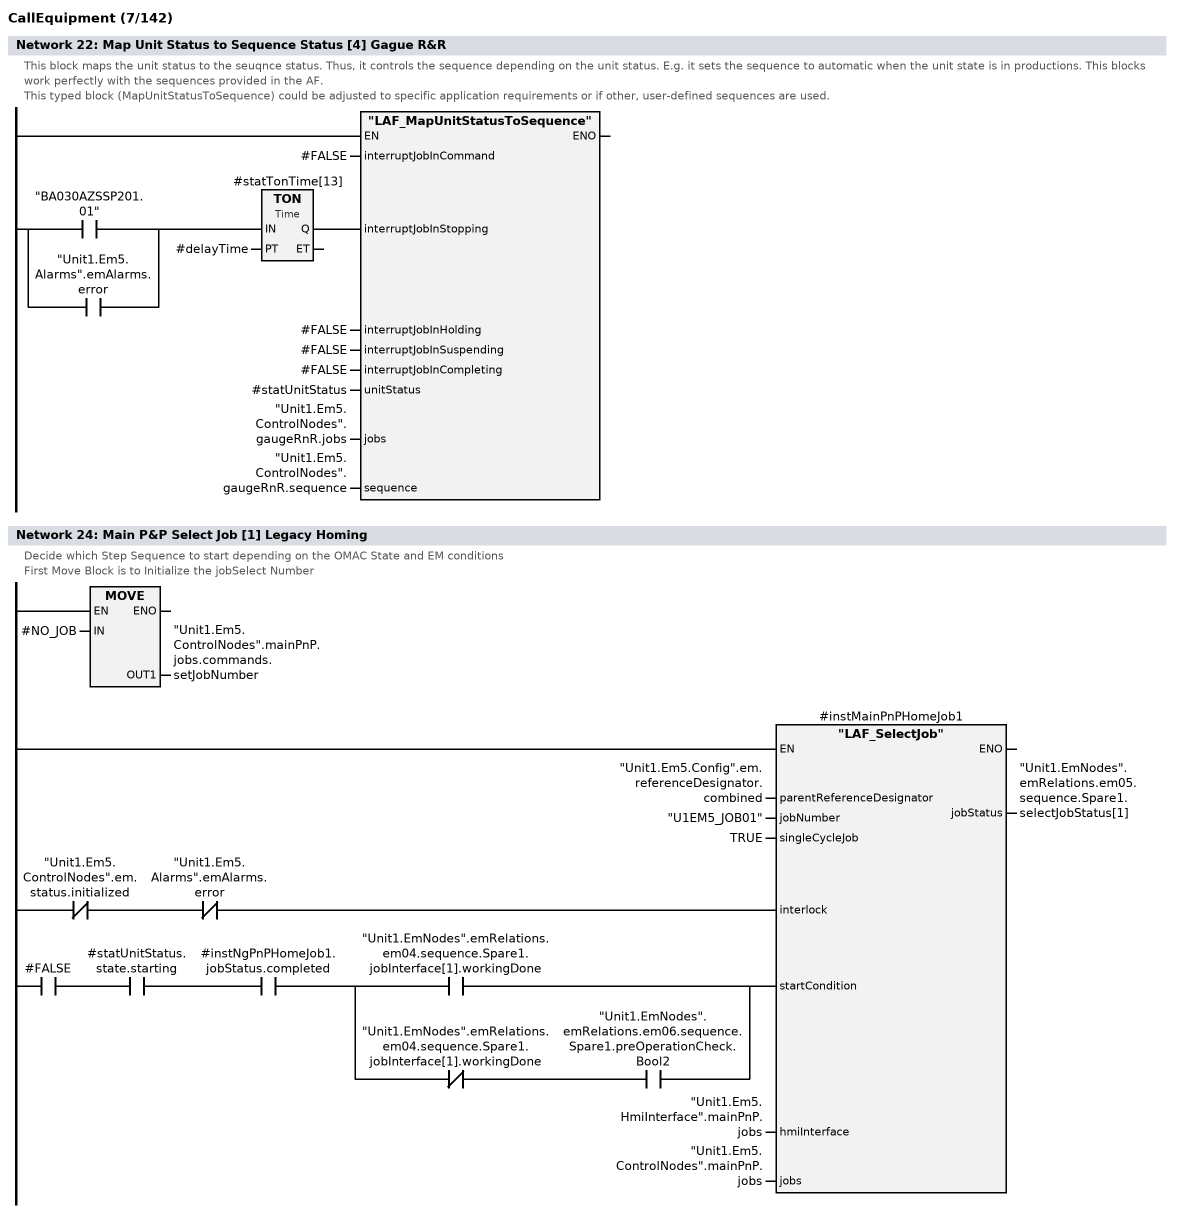
   RUNG wire#powerrail
      "LAF_MapUnitStatusToSequence"(interruptJobInStopping := wire#w2, interruptJobInCommand := #FALSE, interruptJobInHolding := #FALSE, interruptJobInSuspending := #FALSE, interruptJobInCompleting := #FALSE, unitStatus := #statUnitStatus, jobs := "Unit1.Em5.ControlNodes".gaugeRnR.jobs, sequence := "Unit1.Em5.ControlNodes".gaugeRnR.sequence)
   END_RUNG
   RUNG wire#powerrail
      Contact( "BA030AZSSP201.01" )
      wire#w1
      { S7_Templates := "time_type := Time" } #statTonTime[13].TON(pt := #delayTime, et =>)
   END_RUNG wire#w2
   RUNG wire#powerrail
      Contact( "Unit1.Em5.Alarms".emAlarms.error )
   END_RUNG wire#w1
   // the same network as SCL:
   #statTonTime[13].TON(IN := "BA030AZSSP201.01" OR "Unit1.Em5.Alarms".emAlarms.error, PT := #delayTime);
   "LAF_MapUnitStatusToSequence"(interruptJobInCommand := #FALSE,
                           interruptJobInStopping := #statTonTime[13].Q,
                           interruptJobInHolding := #FALSE,
                           interruptJobInSuspending := #FALSE,
                           interruptJobInCompleting := #FALSE,
                           unitStatus := #statUnitStatus,
                           jobs := "Unit1.Em5.ControlNodes".gaugeRnR.jobs,
                           sequence := "Unit1.Em5.ControlNodes".gaugeRnR.sequence);
END_REGION

REGION Network 24: Main P&P Select Job [1] Legacy Homing
   // Decide which Step Sequence to start depending on the OMAC State and EM conditions
   // First Move Block is to Initialize the jobSelect Number
   RUNG wire#powerrail
      Move(in := #NO_JOB, out1 => "Unit1.Em5.ControlNodes".mainPnP.jobs.commands.setJobNumber)
   END_RUNG
   RUNG wire#powerrail
      #instMainPnPHomeJob1(interlock := wire#w1, startCondition := wire#w3, parentReferenceDesignator := "Unit1.Em5.Config".em.referenceDesignator.combined, jobNumber := "U1EM5_JOB01", singleCycleJob := TRUE, hmiInterface := "Unit1.Em5.HmiInterface".mainPnP.jobs, jobs := "Unit1.Em5.ControlNodes".mainPnP.jobs, jobStatus => "Unit1.EmNodes".emRelations.em05.sequence.Spare1.selectJobStatus[1])
   END_RUNG
   RUNG wire#powerrail
      I_Contact( "Unit1.Em5.ControlNodes".em.status.initialized )
      I_Contact( "Unit1.Em5.Alarms".emAlarms.error )
   END_RUNG wire#w1
   RUNG wire#powerrail
      Contact( #FALSE )
      Contact( #statUnitStatus.state.starting )
      Contact( #instNgPnPHomeJob1.jobStatus.completed )
      wire#w2
      Contact( "Unit1.EmNodes".emRelations.em04.sequence.Spare1.jobInterface[1].workingDone )
   END_RUNG wire#w3
   RUNG wire#w2
      I_Contact( "Unit1.EmNodes".emRelations.em04.sequence.Spare1.jobInterface[1].workingDone )
      Contact( "Unit1.EmNodes".emRelations.em06.sequence.Spare1.preOperationCheck.Bool2 )
   END_RUNG wire#w3
   // the same network as SCL:
   "Unit1.Em5.ControlNodes".mainPnP.jobs.commands.setJobNumber := #NO_JOB;
   #instMainPnPHomeJob1(parentReferenceDesignator := "Unit1.Em5.Config".em.referenceDesignator.combined,   // "LAF_SelectJob"
                        jobNumber := "U1EM5_JOB01",
                        singleCycleJob := TRUE,
                        interlock := NOT "Unit1.Em5.ControlNodes".em.status.initialized AND NOT "Unit1.Em5.Alarms".emAlarms.error,
                        startCondition := #FALSE AND #statUnitStatus.state.starting AND #instNgPnPHomeJob1.jobStatus.completed AND ("Unit1.EmNodes".emRelations.em04.sequence.Spare1.jobInterface[1].workingDone OR (NOT "Unit1.EmNodes".emRelations.em04.sequence.Spare1.jobInterface[1].workingDone AND "Unit1.EmNodes".emRelations.em06.sequence.Spare1.preOperationCheck.Bool2)),
                        hmiInterface := "Unit1.Em5.HmiInterface".mainPnP.jobs,
                        jobs := "Unit1.Em5.ControlNodes".mainPnP.jobs,
                        jobStatus => "Unit1.EmNodes".emRelations.em05.sequence.Spare1.selectJobStatus[1]);
END_REGION

REGION Network 25: Main P&P Select Job [10] Homing
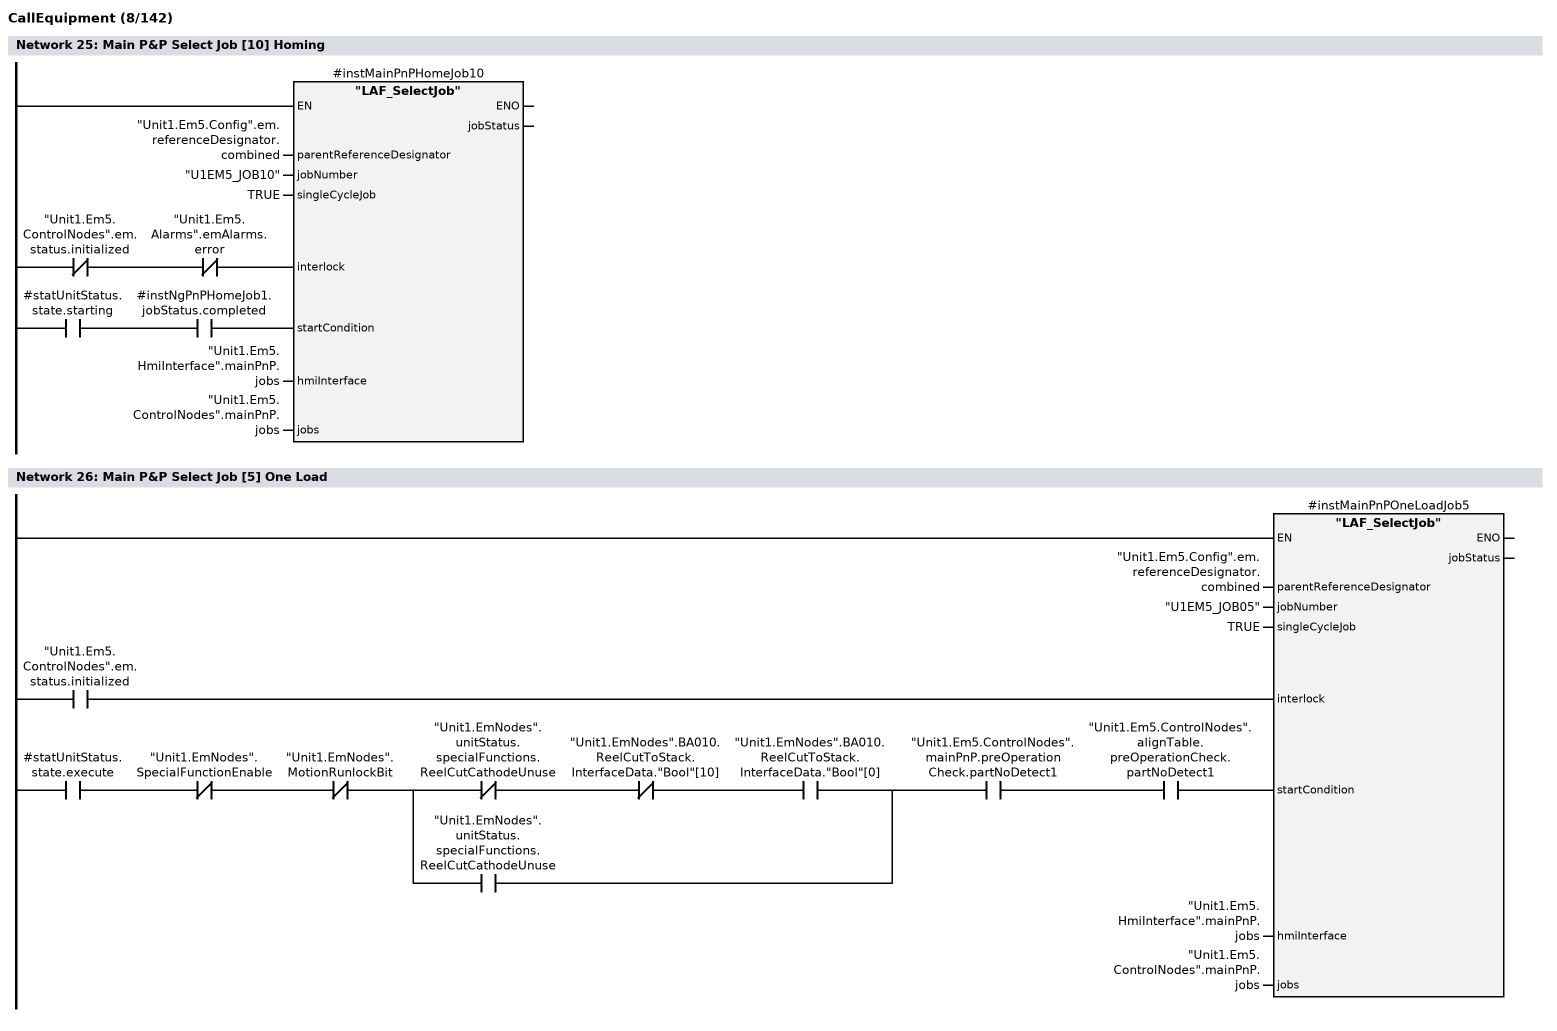
   RUNG wire#powerrail
      #instMainPnPHomeJob10(interlock := wire#w1, startCondition := wire#w2, parentReferenceDesignator := "Unit1.Em5.Config".em.referenceDesignator.combined, jobNumber := "U1EM5_JOB10", singleCycleJob := TRUE, hmiInterface := "Unit1.Em5.HmiInterface".mainPnP.jobs, jobs := "Unit1.Em5.ControlNodes".mainPnP.jobs, jobStatus =>)
   END_RUNG
   RUNG wire#powerrail
      I_Contact( "Unit1.Em5.ControlNodes".em.status.initialized )
      I_Contact( "Unit1.Em5.Alarms".emAlarms.error )
   END_RUNG wire#w1
   RUNG wire#powerrail
      Contact( #statUnitStatus.state.starting )
      Contact( #instNgPnPHomeJob1.jobStatus.completed )
   END_RUNG wire#w2
   // the same network as SCL:
   #instMainPnPHomeJob10(parentReferenceDesignator := "Unit1.Em5.Config".em.referenceDesignator.combined,   // "LAF_SelectJob"
                         jobNumber := "U1EM5_JOB10",
                         singleCycleJob := TRUE,
                         interlock := NOT "Unit1.Em5.ControlNodes".em.status.initialized AND NOT "Unit1.Em5.Alarms".emAlarms.error,
                         startCondition := #statUnitStatus.state.starting AND #instNgPnPHomeJob1.jobStatus.completed,
                         hmiInterface := "Unit1.Em5.HmiInterface".mainPnP.jobs,
                         jobs := "Unit1.Em5.ControlNodes".mainPnP.jobs);
END_REGION

REGION Network 26: Main P&P Select Job [5] One Load
   RUNG wire#powerrail
      #instMainPnPOneLoadJob5(interlock := wire#w1, startCondition := wire#w4, parentReferenceDesignator := "Unit1.Em5.Config".em.referenceDesignator.combined, jobNumber := "U1EM5_JOB05", singleCycleJob := TRUE, hmiInterface := "Unit1.Em5.HmiInterface".mainPnP.jobs, jobs := "Unit1.Em5.ControlNodes".mainPnP.jobs, jobStatus =>)
   END_RUNG
   RUNG wire#powerrail
      Contact( "Unit1.Em5.ControlNodes".em.status.initialized )
   END_RUNG wire#w1
   RUNG wire#powerrail
      Contact( #statUnitStatus.state.execute )
      I_Contact( "Unit1.EmNodes".SpecialFunctionEnable )
      I_Contact( "Unit1.EmNodes".MotionRunlockBit )
      wire#w2
      I_Contact( "Unit1.EmNodes".unitStatus.specialFunctions.ReelCutCathodeUnuse )
      I_Contact( "Unit1.EmNodes".BA010.ReelCutToStack.InterfaceData."Bool"[10] )
      Contact( "Unit1.EmNodes".BA010.ReelCutToStack.InterfaceData."Bool"[0] )
      wire#w3
      Contact( "Unit1.Em5.ControlNodes".mainPnP.preOperationCheck.partNoDetect1 )
      Contact( "Unit1.Em5.ControlNodes".alignTable.preOperationCheck.partNoDetect1 )
   END_RUNG wire#w4
   RUNG wire#w2
      Contact( "Unit1.EmNodes".unitStatus.specialFunctions.ReelCutCathodeUnuse )
   END_RUNG wire#w3
   // the same network as SCL:
   #instMainPnPOneLoadJob5(parentReferenceDesignator := "Unit1.Em5.Config".em.referenceDesignator.combined,   // "LAF_SelectJob"
                           jobNumber := "U1EM5_JOB05",
                           singleCycleJob := TRUE,
                           interlock := "Unit1.Em5.ControlNodes".em.status.initialized,
                           startCondition := #statUnitStatus.state.execute AND NOT "Unit1.EmNodes".SpecialFunctionEnable AND NOT "Unit1.EmNodes".MotionRunlockBit AND ((NOT "Unit1.EmNodes".unitStatus.specialFunctions.ReelCutCathodeUnuse AND NOT "Unit1.EmNodes".BA010.ReelCutToStack.InterfaceData."Bool"[10] AND "Unit1.EmNodes".BA010.ReelCutToStack.InterfaceData."Bool"[0]) OR "Unit1.EmNodes".unitStatus.specialFunctions.ReelCutCathodeUnuse) AND "Unit1.Em5.ControlNodes".mainPnP.preOperationCheck.partNoDetect1 AND "Unit1.Em5.ControlNodes".alignTable.preOperationCheck.partNoDetect1,
                           hmiInterface := "Unit1.Em5.HmiInterface".mainPnP.jobs,
                           jobs := "Unit1.Em5.ControlNodes".mainPnP.jobs);
END_REGION

REGION Network 27: Main P&P Select Job [6] One UnLoad
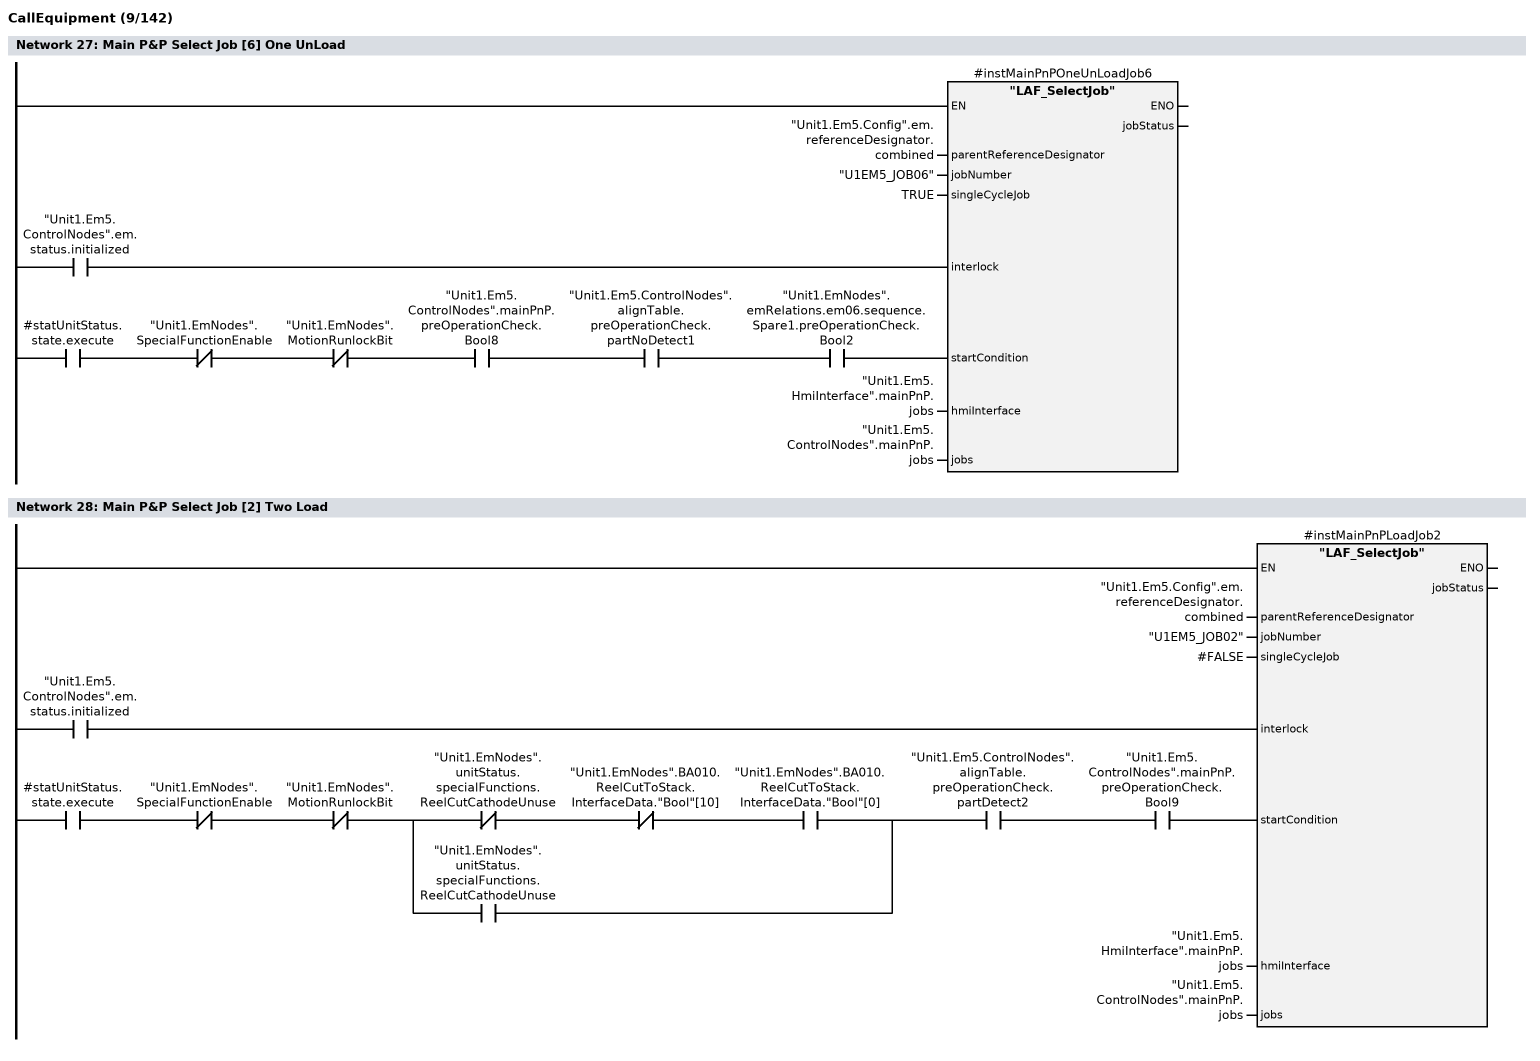
   RUNG wire#powerrail
      #instMainPnPOneUnLoadJob6(interlock := wire#w1, startCondition := wire#w2, parentReferenceDesignator := "Unit1.Em5.Config".em.referenceDesignator.combined, jobNumber := "U1EM5_JOB06", singleCycleJob := TRUE, hmiInterface := "Unit1.Em5.HmiInterface".mainPnP.jobs, jobs := "Unit1.Em5.ControlNodes".mainPnP.jobs, jobStatus =>)
   END_RUNG
   RUNG wire#powerrail
      Contact( "Unit1.Em5.ControlNodes".em.status.initialized )
   END_RUNG wire#w1
   RUNG wire#powerrail
      Contact( #statUnitStatus.state.execute )
      I_Contact( "Unit1.EmNodes".SpecialFunctionEnable )
      I_Contact( "Unit1.EmNodes".MotionRunlockBit )
      Contact( "Unit1.Em5.ControlNodes".mainPnP.preOperationCheck.Bool8 )
      Contact( "Unit1.Em5.ControlNodes".alignTable.preOperationCheck.partNoDetect1 )
      Contact( "Unit1.EmNodes".emRelations.em06.sequence.Spare1.preOperationCheck.Bool2 )
   END_RUNG wire#w2
   // the same network as SCL:
   #instMainPnPOneUnLoadJob6(parentReferenceDesignator := "Unit1.Em5.Config".em.referenceDesignator.combined,   // "LAF_SelectJob"
                           jobNumber := "U1EM5_JOB06",
                           singleCycleJob := TRUE,
                           interlock := "Unit1.Em5.ControlNodes".em.status.initialized,
                           startCondition := #statUnitStatus.state.execute AND NOT "Unit1.EmNodes".SpecialFunctionEnable AND NOT "Unit1.EmNodes".MotionRunlockBit AND "Unit1.Em5.ControlNodes".mainPnP.preOperationCheck.Bool8 AND "Unit1.Em5.ControlNodes".alignTable.preOperationCheck.partNoDetect1 AND "Unit1.EmNodes".emRelations.em06.sequence.Spare1.preOperationCheck.Bool2,
                           hmiInterface := "Unit1.Em5.HmiInterface".mainPnP.jobs,
                           jobs := "Unit1.Em5.ControlNodes".mainPnP.jobs);
END_REGION

REGION Network 28: Main P&P Select Job [2] Two Load
   RUNG wire#powerrail
      #instMainPnPLoadJob2(interlock := wire#w1, startCondition := wire#w4, parentReferenceDesignator := "Unit1.Em5.Config".em.referenceDesignator.combined, jobNumber := "U1EM5_JOB02", singleCycleJob := #FALSE, hmiInterface := "Unit1.Em5.HmiInterface".mainPnP.jobs, jobs := "Unit1.Em5.ControlNodes".mainPnP.jobs, jobStatus =>)
   END_RUNG
   RUNG wire#powerrail
      Contact( "Unit1.Em5.ControlNodes".em.status.initialized )
   END_RUNG wire#w1
   RUNG wire#powerrail
      Contact( #statUnitStatus.state.execute )
      I_Contact( "Unit1.EmNodes".SpecialFunctionEnable )
      I_Contact( "Unit1.EmNodes".MotionRunlockBit )
      wire#w2
      I_Contact( "Unit1.EmNodes".unitStatus.specialFunctions.ReelCutCathodeUnuse )
      I_Contact( "Unit1.EmNodes".BA010.ReelCutToStack.InterfaceData."Bool"[10] )
      Contact( "Unit1.EmNodes".BA010.ReelCutToStack.InterfaceData."Bool"[0] )
      wire#w3
      Contact( "Unit1.Em5.ControlNodes".alignTable.preOperationCheck.partDetect2 )
      Contact( "Unit1.Em5.ControlNodes".mainPnP.preOperationCheck.Bool9 )
   END_RUNG wire#w4
   RUNG wire#w2
      Contact( "Unit1.EmNodes".unitStatus.specialFunctions.ReelCutCathodeUnuse )
   END_RUNG wire#w3
   // the same network as SCL:
   #instMainPnPLoadJob2(parentReferenceDesignator := "Unit1.Em5.Config".em.referenceDesignator.combined,   // "LAF_SelectJob"
                        jobNumber := "U1EM5_JOB02",
                        singleCycleJob := #FALSE,
                        interlock := "Unit1.Em5.ControlNodes".em.status.initialized,
                        startCondition := #statUnitStatus.state.execute AND NOT "Unit1.EmNodes".SpecialFunctionEnable AND NOT "Unit1.EmNodes".MotionRunlockBit AND ((NOT "Unit1.EmNodes".unitStatus.specialFunctions.ReelCutCathodeUnuse AND NOT "Unit1.EmNodes".BA010.ReelCutToStack.InterfaceData."Bool"[10] AND "Unit1.EmNodes".BA010.ReelCutToStack.InterfaceData."Bool"[0]) OR "Unit1.EmNodes".unitStatus.specialFunctions.ReelCutCathodeUnuse) AND "Unit1.Em5.ControlNodes".alignTable.preOperationCheck.partDetect2 AND "Unit1.Em5.ControlNodes".mainPnP.preOperationCheck.Bool9,
                        hmiInterface := "Unit1.Em5.HmiInterface".mainPnP.jobs,
                        jobs := "Unit1.Em5.ControlNodes".mainPnP.jobs);
END_REGION

REGION Network 29: Main P&P Select Job [3] Two UnLoad
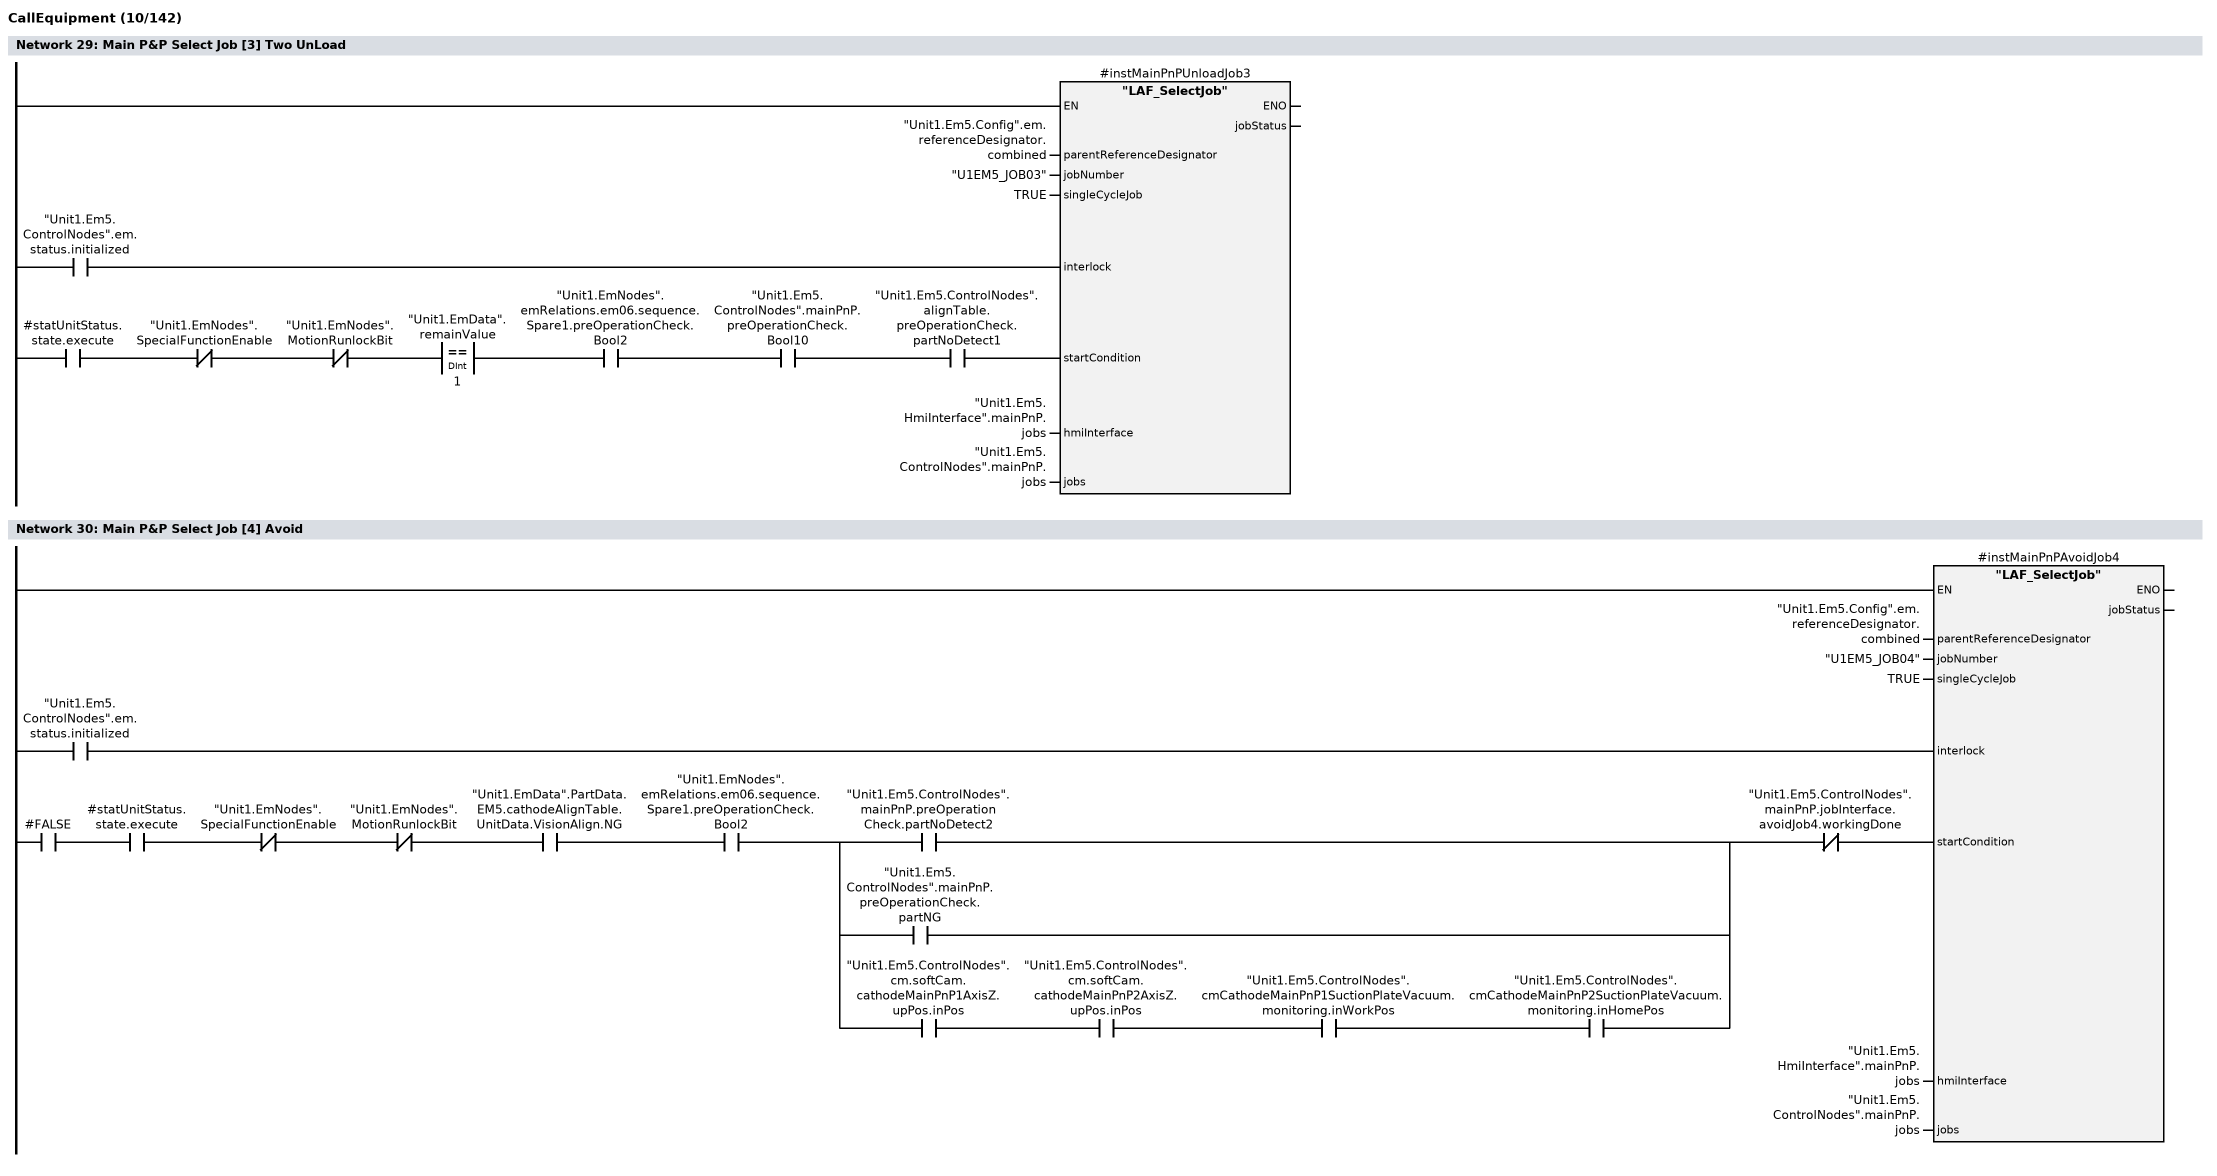
   RUNG wire#powerrail
      #instMainPnPUnloadJob3(interlock := wire#w1, startCondition := wire#w2, parentReferenceDesignator := "Unit1.Em5.Config".em.referenceDesignator.combined, jobNumber := "U1EM5_JOB03", singleCycleJob := TRUE, hmiInterface := "Unit1.Em5.HmiInterface".mainPnP.jobs, jobs := "Unit1.Em5.ControlNodes".mainPnP.jobs, jobStatus =>)
   END_RUNG
   RUNG wire#powerrail
      Contact( "Unit1.Em5.ControlNodes".em.status.initialized )
   END_RUNG wire#w1
   RUNG wire#powerrail
      Contact( #statUnitStatus.state.execute )
      I_Contact( "Unit1.EmNodes".SpecialFunctionEnable )
      I_Contact( "Unit1.EmNodes".MotionRunlockBit )
      { S7_Templates := "SrcType := DInt" } EQ_Contact(in1 := "Unit1.EmData".remainValue, in2 := 1)
      Contact( "Unit1.EmNodes".emRelations.em06.sequence.Spare1.preOperationCheck.Bool2 )
      Contact( "Unit1.Em5.ControlNodes".mainPnP.preOperationCheck.Bool10 )
      Contact( "Unit1.Em5.ControlNodes".alignTable.preOperationCheck.partNoDetect1 )
   END_RUNG wire#w2
   // the same network as SCL:
   #instMainPnPUnloadJob3(parentReferenceDesignator := "Unit1.Em5.Config".em.referenceDesignator.combined,   // "LAF_SelectJob"
                          jobNumber := "U1EM5_JOB03",
                          singleCycleJob := TRUE,
                          interlock := "Unit1.Em5.ControlNodes".em.status.initialized,
                          startCondition := #statUnitStatus.state.execute AND NOT "Unit1.EmNodes".SpecialFunctionEnable AND NOT "Unit1.EmNodes".MotionRunlockBit AND ("Unit1.EmData".remainValue = 1) AND "Unit1.EmNodes".emRelations.em06.sequence.Spare1.preOperationCheck.Bool2 AND "Unit1.Em5.ControlNodes".mainPnP.preOperationCheck.Bool10 AND "Unit1.Em5.ControlNodes".alignTable.preOperationCheck.partNoDetect1,
                          hmiInterface := "Unit1.Em5.HmiInterface".mainPnP.jobs,
                          jobs := "Unit1.Em5.ControlNodes".mainPnP.jobs);
END_REGION

REGION Network 30: Main P&P Select Job [4] Avoid
   RUNG wire#powerrail
      #instMainPnPAvoidJob4(interlock := wire#w1, startCondition := wire#w4, parentReferenceDesignator := "Unit1.Em5.Config".em.referenceDesignator.combined, jobNumber := "U1EM5_JOB04", singleCycleJob := TRUE, hmiInterface := "Unit1.Em5.HmiInterface".mainPnP.jobs, jobs := "Unit1.Em5.ControlNodes".mainPnP.jobs, jobStatus =>)
   END_RUNG
   RUNG wire#powerrail
      Contact( "Unit1.Em5.ControlNodes".em.status.initialized )
   END_RUNG wire#w1
   RUNG wire#powerrail
      Contact( #FALSE )
      Contact( #statUnitStatus.state.execute )
      I_Contact( "Unit1.EmNodes".SpecialFunctionEnable )
      I_Contact( "Unit1.EmNodes".MotionRunlockBit )
      Contact( "Unit1.EmData".PartData.EM5.cathodeAlignTable.UnitData.VisionAlign.NG )
      Contact( "Unit1.EmNodes".emRelations.em06.sequence.Spare1.preOperationCheck.Bool2 )
      wire#w2
      Contact( "Unit1.Em5.ControlNodes".mainPnP.preOperationCheck.partNoDetect2 )
      wire#w3
      I_Contact( "Unit1.Em5.ControlNodes".mainPnP.jobInterface.avoidJob4.workingDone )
   END_RUNG wire#w4
   RUNG wire#w2
      Contact( "Unit1.Em5.ControlNodes".mainPnP.preOperationCheck.partNG )
   END_RUNG wire#w3
   RUNG wire#w2
      Contact( "Unit1.Em5.ControlNodes".cm.softCam.cathodeMainPnP1AxisZ.upPos.inPos )
      Contact( "Unit1.Em5.ControlNodes".cm.softCam.cathodeMainPnP2AxisZ.upPos.inPos )
      Contact( "Unit1.Em5.ControlNodes".cmCathodeMainPnP1SuctionPlateVacuum.monitoring.inWorkPos )
      Contact( "Unit1.Em5.ControlNodes".cmCathodeMainPnP2SuctionPlateVacuum.monitoring.inHomePos )
   END_RUNG wire#w3
   // the same network as SCL:
   #instMainPnPAvoidJob4(parentReferenceDesignator := "Unit1.Em5.Config".em.referenceDesignator.combined,   // "LAF_SelectJob"
                         jobNumber := "U1EM5_JOB04",
                         singleCycleJob := TRUE,
                         interlock := "Unit1.Em5.ControlNodes".em.status.initialized,
                         startCondition := #FALSE AND #statUnitStatus.state.execute AND NOT "Unit1.EmNodes".SpecialFunctionEnable AND NOT "Unit1.EmNodes".MotionRunlockBit AND "Unit1.EmData".PartData.EM5.cathodeAlignTable.UnitData.VisionAlign.NG AND "Unit1.EmNodes".emRelations.em06.sequence.Spare1.preOperationCheck.Bool2 AND ("Unit1.Em5.ControlNodes".mainPnP.preOperationCheck.partNoDetect2 OR "Unit1.Em5.ControlNodes".mainPnP.preOperationCheck.partNG OR ("Unit1.Em5.ControlNodes".cm.softCam.cathodeMainPnP1AxisZ.upPos.inPos AND "Unit1.Em5.ControlNodes".cm.softCam.cathodeMainPnP2AxisZ.upPos.inPos AND "Unit1.Em5.ControlNodes".cmCathodeMainPnP1SuctionPlateVacuum.monitoring.inWorkPos AND "Unit1.Em5.ControlNodes".cmCathodeMainPnP2SuctionPlateVacuum.monitoring.inHomePos)) AND NOT "Unit1.Em5.ControlNodes".mainPnP.jobInterface.avoidJob4.workingDone,
                         hmiInterface := "Unit1.Em5.HmiInterface".mainPnP.jobs,
                         jobs := "Unit1.Em5.ControlNodes".mainPnP.jobs);
END_REGION

REGION Network 32: Main P&P Job Interface [10] Homing
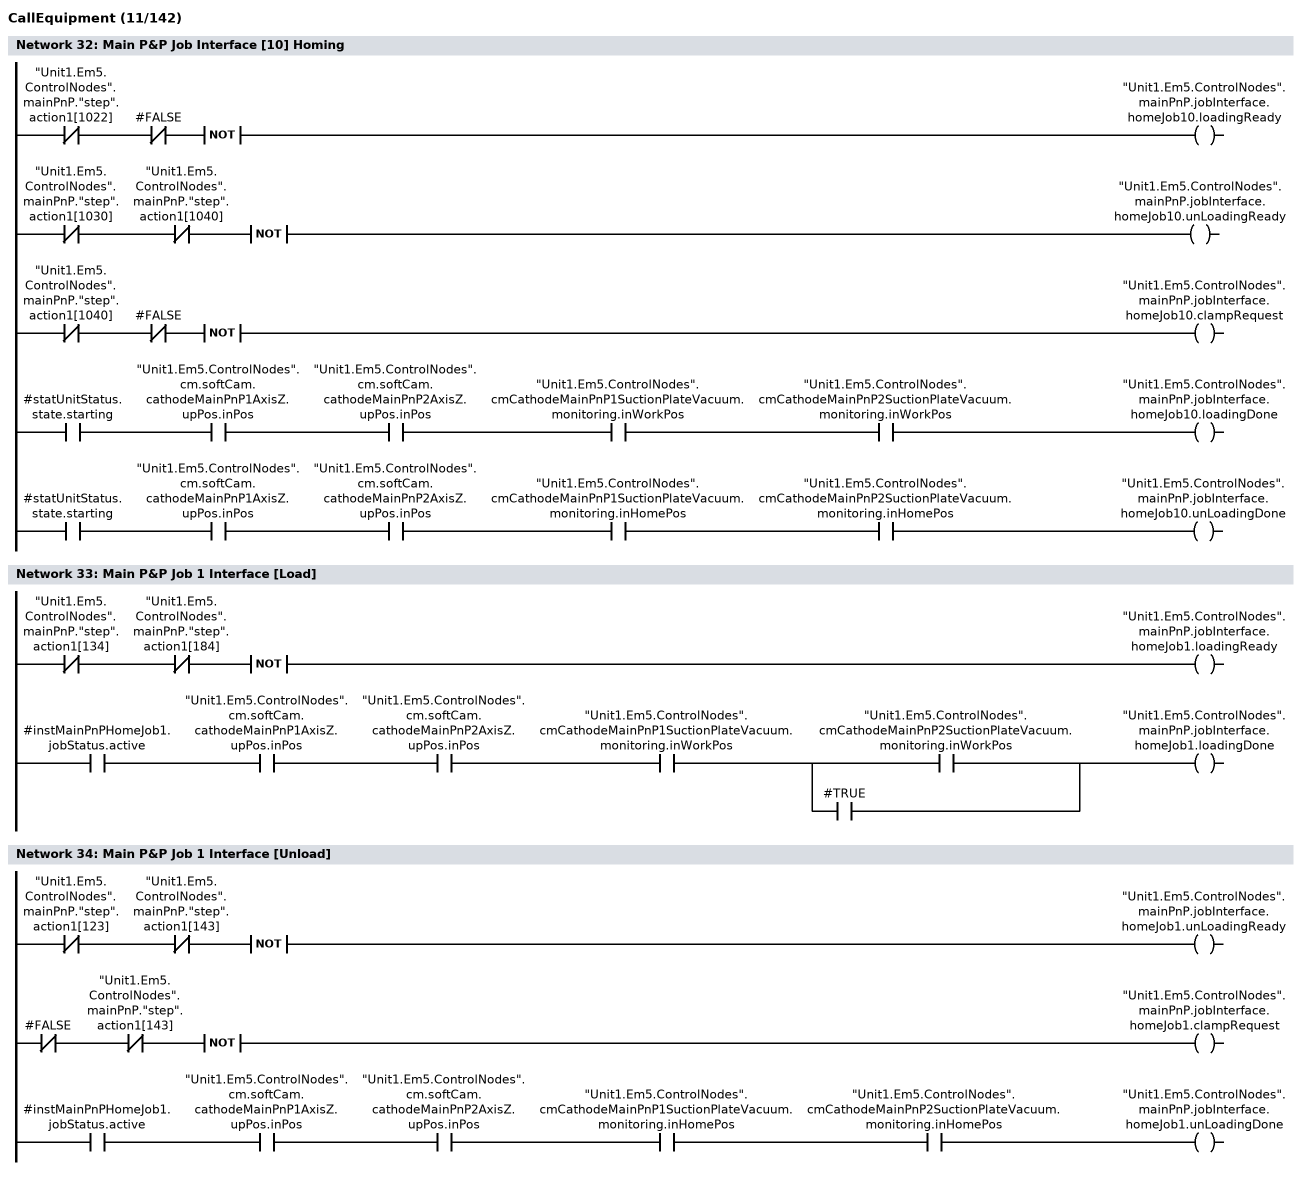
   RUNG wire#powerrail
      I_Contact( "Unit1.Em5.ControlNodes".mainPnP."step".action1[1022] )
      I_Contact( #FALSE )
      Not()
      Coil( "Unit1.Em5.ControlNodes".mainPnP.jobInterface.homeJob10.loadingReady )
   END_RUNG
   RUNG wire#powerrail
      I_Contact( "Unit1.Em5.ControlNodes".mainPnP."step".action1[1030] )
      I_Contact( "Unit1.Em5.ControlNodes".mainPnP."step".action1[1040] )
      Not()
      Coil( "Unit1.Em5.ControlNodes".mainPnP.jobInterface.homeJob10.unLoadingReady )
   END_RUNG
   RUNG wire#powerrail
      I_Contact( "Unit1.Em5.ControlNodes".mainPnP."step".action1[1040] )
      I_Contact( #FALSE )
      Not()
      Coil( "Unit1.Em5.ControlNodes".mainPnP.jobInterface.homeJob10.clampRequest )
   END_RUNG
   RUNG wire#powerrail
      Contact( #statUnitStatus.state.starting )
      Contact( "Unit1.Em5.ControlNodes".cm.softCam.cathodeMainPnP1AxisZ.upPos.inPos )
      Contact( "Unit1.Em5.ControlNodes".cm.softCam.cathodeMainPnP2AxisZ.upPos.inPos )
      Contact( "Unit1.Em5.ControlNodes".cmCathodeMainPnP1SuctionPlateVacuum.monitoring.inWorkPos )
      Contact( "Unit1.Em5.ControlNodes".cmCathodeMainPnP2SuctionPlateVacuum.monitoring.inWorkPos )
      Coil( "Unit1.Em5.ControlNodes".mainPnP.jobInterface.homeJob10.loadingDone )
   END_RUNG
   RUNG wire#powerrail
      Contact( #statUnitStatus.state.starting )
      Contact( "Unit1.Em5.ControlNodes".cm.softCam.cathodeMainPnP1AxisZ.upPos.inPos )
      Contact( "Unit1.Em5.ControlNodes".cm.softCam.cathodeMainPnP2AxisZ.upPos.inPos )
      Contact( "Unit1.Em5.ControlNodes".cmCathodeMainPnP1SuctionPlateVacuum.monitoring.inHomePos )
      Contact( "Unit1.Em5.ControlNodes".cmCathodeMainPnP2SuctionPlateVacuum.monitoring.inHomePos )
      Coil( "Unit1.Em5.ControlNodes".mainPnP.jobInterface.homeJob10.unLoadingDone )
   END_RUNG
   // the same network as SCL:
   "Unit1.Em5.ControlNodes".mainPnP.jobInterface.homeJob10.loadingReady := NOT (NOT "Unit1.Em5.ControlNodes".mainPnP."step".action1[1022] AND NOT #FALSE);
   "Unit1.Em5.ControlNodes".mainPnP.jobInterface.homeJob10.unLoadingReady := NOT (NOT "Unit1.Em5.ControlNodes".mainPnP."step".action1[1030] AND NOT "Unit1.Em5.ControlNodes".mainPnP."step".action1[1040]);
   "Unit1.Em5.ControlNodes".mainPnP.jobInterface.homeJob10.clampRequest := NOT (NOT "Unit1.Em5.ControlNodes".mainPnP."step".action1[1040] AND NOT #FALSE);
   "Unit1.Em5.ControlNodes".mainPnP.jobInterface.homeJob10.loadingDone := #statUnitStatus.state.starting AND "Unit1.Em5.ControlNodes".cm.softCam.cathodeMainPnP1AxisZ.upPos.inPos AND "Unit1.Em5.ControlNodes".cm.softCam.cathodeMainPnP2AxisZ.upPos.inPos AND "Unit1.Em5.ControlNodes".cmCathodeMainPnP1SuctionPlateVacuum.monitoring.inWorkPos AND "Unit1.Em5.ControlNodes".cmCathodeMainPnP2SuctionPlateVacuum.monitoring.inWorkPos;
   "Unit1.Em5.ControlNodes".mainPnP.jobInterface.homeJob10.unLoadingDone := #statUnitStatus.state.starting AND "Unit1.Em5.ControlNodes".cm.softCam.cathodeMainPnP1AxisZ.upPos.inPos AND "Unit1.Em5.ControlNodes".cm.softCam.cathodeMainPnP2AxisZ.upPos.inPos AND "Unit1.Em5.ControlNodes".cmCathodeMainPnP1SuctionPlateVacuum.monitoring.inHomePos AND "Unit1.Em5.ControlNodes".cmCathodeMainPnP2SuctionPlateVacuum.monitoring.inHomePos;
END_REGION

REGION Network 33: Main P&P Job 1 Interface [Load]
   RUNG wire#powerrail
      I_Contact( "Unit1.Em5.ControlNodes".mainPnP."step".action1[134] )
      I_Contact( "Unit1.Em5.ControlNodes".mainPnP."step".action1[184] )
      Not()
      Coil( "Unit1.Em5.ControlNodes".mainPnP.jobInterface.homeJob1.loadingReady )
   END_RUNG
   RUNG wire#powerrail
      Contact( #instMainPnPHomeJob1.jobStatus.active )
      Contact( "Unit1.Em5.ControlNodes".cm.softCam.cathodeMainPnP1AxisZ.upPos.inPos )
      Contact( "Unit1.Em5.ControlNodes".cm.softCam.cathodeMainPnP2AxisZ.upPos.inPos )
      Contact( "Unit1.Em5.ControlNodes".cmCathodeMainPnP1SuctionPlateVacuum.monitoring.inWorkPos )
      wire#w1
      Contact( "Unit1.Em5.ControlNodes".cmCathodeMainPnP2SuctionPlateVacuum.monitoring.inWorkPos )
      wire#w2
      Coil( "Unit1.Em5.ControlNodes".mainPnP.jobInterface.homeJob1.loadingDone )
   END_RUNG
   RUNG wire#w1
      Contact( #TRUE )
   END_RUNG wire#w2
   // the same network as SCL:
   "Unit1.Em5.ControlNodes".mainPnP.jobInterface.homeJob1.loadingReady := NOT (NOT "Unit1.Em5.ControlNodes".mainPnP."step".action1[134] AND NOT "Unit1.Em5.ControlNodes".mainPnP."step".action1[184]);
   "Unit1.Em5.ControlNodes".mainPnP.jobInterface.homeJob1.loadingDone := #instMainPnPHomeJob1.jobStatus.active AND "Unit1.Em5.ControlNodes".cm.softCam.cathodeMainPnP1AxisZ.upPos.inPos AND "Unit1.Em5.ControlNodes".cm.softCam.cathodeMainPnP2AxisZ.upPos.inPos AND "Unit1.Em5.ControlNodes".cmCathodeMainPnP1SuctionPlateVacuum.monitoring.inWorkPos AND ("Unit1.Em5.ControlNodes".cmCathodeMainPnP2SuctionPlateVacuum.monitoring.inWorkPos OR #TRUE);
END_REGION

REGION Network 34: Main P&P Job 1 Interface [Unload]
   RUNG wire#powerrail
      I_Contact( "Unit1.Em5.ControlNodes".mainPnP."step".action1[123] )
      I_Contact( "Unit1.Em5.ControlNodes".mainPnP."step".action1[143] )
      Not()
      Coil( "Unit1.Em5.ControlNodes".mainPnP.jobInterface.homeJob1.unLoadingReady )
   END_RUNG
   RUNG wire#powerrail
      I_Contact( #FALSE )
      I_Contact( "Unit1.Em5.ControlNodes".mainPnP."step".action1[143] )
      Not()
      Coil( "Unit1.Em5.ControlNodes".mainPnP.jobInterface.homeJob1.clampRequest )
   END_RUNG
   RUNG wire#powerrail
      Contact( #instMainPnPHomeJob1.jobStatus.active )
      Contact( "Unit1.Em5.ControlNodes".cm.softCam.cathodeMainPnP1AxisZ.upPos.inPos )
      Contact( "Unit1.Em5.ControlNodes".cm.softCam.cathodeMainPnP2AxisZ.upPos.inPos )
      Contact( "Unit1.Em5.ControlNodes".cmCathodeMainPnP1SuctionPlateVacuum.monitoring.inHomePos )
      Contact( "Unit1.Em5.ControlNodes".cmCathodeMainPnP2SuctionPlateVacuum.monitoring.inHomePos )
      Coil( "Unit1.Em5.ControlNodes".mainPnP.jobInterface.homeJob1.unLoadingDone )
   END_RUNG
   // the same network as SCL:
   "Unit1.Em5.ControlNodes".mainPnP.jobInterface.homeJob1.unLoadingReady := NOT (NOT "Unit1.Em5.ControlNodes".mainPnP."step".action1[123] AND NOT "Unit1.Em5.ControlNodes".mainPnP."step".action1[143]);
   "Unit1.Em5.ControlNodes".mainPnP.jobInterface.homeJob1.clampRequest := NOT (NOT #FALSE AND NOT "Unit1.Em5.ControlNodes".mainPnP."step".action1[143]);
   "Unit1.Em5.ControlNodes".mainPnP.jobInterface.homeJob1.unLoadingDone := #instMainPnPHomeJob1.jobStatus.active AND "Unit1.Em5.ControlNodes".cm.softCam.cathodeMainPnP1AxisZ.upPos.inPos AND "Unit1.Em5.ControlNodes".cm.softCam.cathodeMainPnP2AxisZ.upPos.inPos AND "Unit1.Em5.ControlNodes".cmCathodeMainPnP1SuctionPlateVacuum.monitoring.inHomePos AND "Unit1.Em5.ControlNodes".cmCathodeMainPnP2SuctionPlateVacuum.monitoring.inHomePos;
END_REGION

REGION Network 35: Main P&P Job 2 Interface [Load]
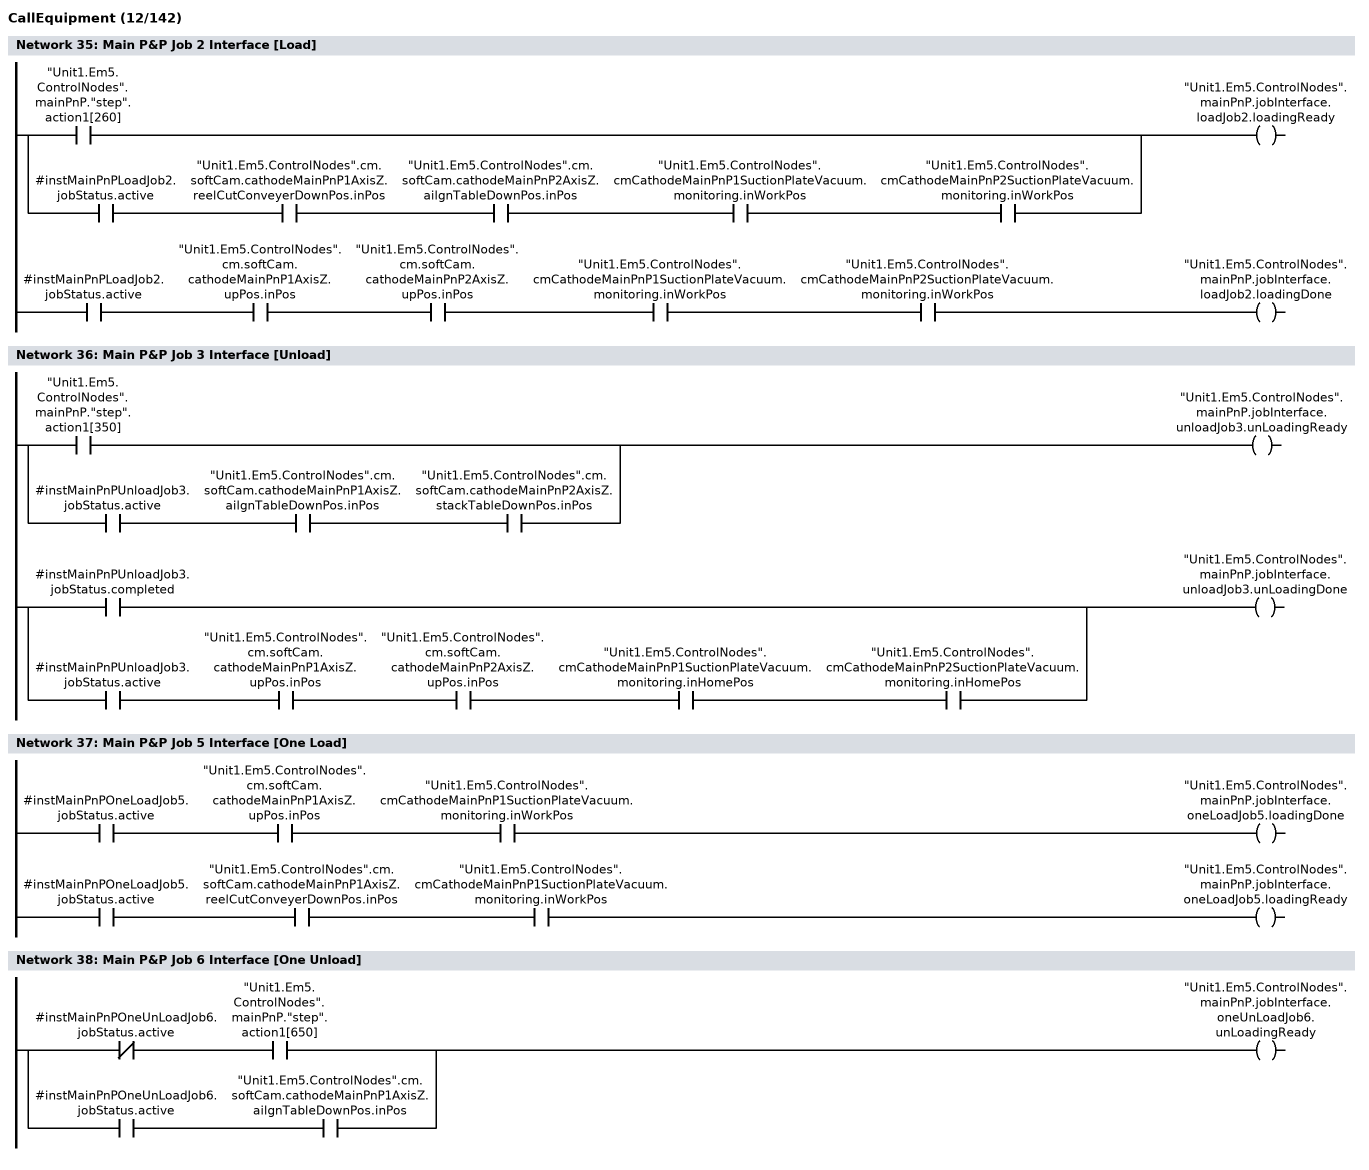
   RUNG wire#powerrail
      Contact( "Unit1.Em5.ControlNodes".mainPnP."step".action1[260] )
      wire#w1
      Coil( "Unit1.Em5.ControlNodes".mainPnP.jobInterface.loadJob2.loadingReady )
   END_RUNG
   RUNG wire#powerrail
      Contact( #instMainPnPLoadJob2.jobStatus.active )
      Contact( "Unit1.Em5.ControlNodes".cm.softCam.cathodeMainPnP1AxisZ.reelCutConveyerDownPos.inPos )
      Contact( "Unit1.Em5.ControlNodes".cm.softCam.cathodeMainPnP2AxisZ.ailgnTableDownPos.inPos )
      Contact( "Unit1.Em5.ControlNodes".cmCathodeMainPnP1SuctionPlateVacuum.monitoring.inWorkPos )
      Contact( "Unit1.Em5.ControlNodes".cmCathodeMainPnP2SuctionPlateVacuum.monitoring.inWorkPos )
   END_RUNG wire#w1
   RUNG wire#powerrail
      Contact( #instMainPnPLoadJob2.jobStatus.active )
      Contact( "Unit1.Em5.ControlNodes".cm.softCam.cathodeMainPnP1AxisZ.upPos.inPos )
      Contact( "Unit1.Em5.ControlNodes".cm.softCam.cathodeMainPnP2AxisZ.upPos.inPos )
      Contact( "Unit1.Em5.ControlNodes".cmCathodeMainPnP1SuctionPlateVacuum.monitoring.inWorkPos )
      Contact( "Unit1.Em5.ControlNodes".cmCathodeMainPnP2SuctionPlateVacuum.monitoring.inWorkPos )
      Coil( "Unit1.Em5.ControlNodes".mainPnP.jobInterface.loadJob2.loadingDone )
   END_RUNG
   // the same network as SCL:
   "Unit1.Em5.ControlNodes".mainPnP.jobInterface.loadJob2.loadingReady := "Unit1.Em5.ControlNodes".mainPnP."step".action1[260] OR (#instMainPnPLoadJob2.jobStatus.active AND "Unit1.Em5.ControlNodes".cm.softCam.cathodeMainPnP1AxisZ.reelCutConveyerDownPos.inPos AND "Unit1.Em5.ControlNodes".cm.softCam.cathodeMainPnP2AxisZ.ailgnTableDownPos.inPos AND "Unit1.Em5.ControlNodes".cmCathodeMainPnP1SuctionPlateVacuum.monitoring.inWorkPos AND "Unit1.Em5.ControlNodes".cmCathodeMainPnP2SuctionPlateVacuum.monitoring.inWorkPos);
   "Unit1.Em5.ControlNodes".mainPnP.jobInterface.loadJob2.loadingDone := #instMainPnPLoadJob2.jobStatus.active AND "Unit1.Em5.ControlNodes".cm.softCam.cathodeMainPnP1AxisZ.upPos.inPos AND "Unit1.Em5.ControlNodes".cm.softCam.cathodeMainPnP2AxisZ.upPos.inPos AND "Unit1.Em5.ControlNodes".cmCathodeMainPnP1SuctionPlateVacuum.monitoring.inWorkPos AND "Unit1.Em5.ControlNodes".cmCathodeMainPnP2SuctionPlateVacuum.monitoring.inWorkPos;
END_REGION

REGION Network 36: Main P&P Job 3 Interface [Unload]
   RUNG wire#powerrail
      Contact( "Unit1.Em5.ControlNodes".mainPnP."step".action1[350] )
      wire#w1
      Coil( "Unit1.Em5.ControlNodes".mainPnP.jobInterface.unloadJob3.unLoadingReady )
   END_RUNG
   RUNG wire#powerrail
      Contact( #instMainPnPUnloadJob3.jobStatus.active )
      Contact( "Unit1.Em5.ControlNodes".cm.softCam.cathodeMainPnP1AxisZ.ailgnTableDownPos.inPos )
      Contact( "Unit1.Em5.ControlNodes".cm.softCam.cathodeMainPnP2AxisZ.stackTableDownPos.inPos )
   END_RUNG wire#w1
   RUNG wire#powerrail
      Contact( #instMainPnPUnloadJob3.jobStatus.completed )
      wire#w2
      Coil( "Unit1.Em5.ControlNodes".mainPnP.jobInterface.unloadJob3.unLoadingDone )
   END_RUNG
   RUNG wire#powerrail
      Contact( #instMainPnPUnloadJob3.jobStatus.active )
      Contact( "Unit1.Em5.ControlNodes".cm.softCam.cathodeMainPnP1AxisZ.upPos.inPos )
      Contact( "Unit1.Em5.ControlNodes".cm.softCam.cathodeMainPnP2AxisZ.upPos.inPos )
      Contact( "Unit1.Em5.ControlNodes".cmCathodeMainPnP1SuctionPlateVacuum.monitoring.inHomePos )
      Contact( "Unit1.Em5.ControlNodes".cmCathodeMainPnP2SuctionPlateVacuum.monitoring.inHomePos )
   END_RUNG wire#w2
   // the same network as SCL:
   "Unit1.Em5.ControlNodes".mainPnP.jobInterface.unloadJob3.unLoadingReady := "Unit1.Em5.ControlNodes".mainPnP."step".action1[350] OR (#instMainPnPUnloadJob3.jobStatus.active AND "Unit1.Em5.ControlNodes".cm.softCam.cathodeMainPnP1AxisZ.ailgnTableDownPos.inPos AND "Unit1.Em5.ControlNodes".cm.softCam.cathodeMainPnP2AxisZ.stackTableDownPos.inPos);
   "Unit1.Em5.ControlNodes".mainPnP.jobInterface.unloadJob3.unLoadingDone := #instMainPnPUnloadJob3.jobStatus.completed OR (#instMainPnPUnloadJob3.jobStatus.active AND "Unit1.Em5.ControlNodes".cm.softCam.cathodeMainPnP1AxisZ.upPos.inPos AND "Unit1.Em5.ControlNodes".cm.softCam.cathodeMainPnP2AxisZ.upPos.inPos AND "Unit1.Em5.ControlNodes".cmCathodeMainPnP1SuctionPlateVacuum.monitoring.inHomePos AND "Unit1.Em5.ControlNodes".cmCathodeMainPnP2SuctionPlateVacuum.monitoring.inHomePos);
END_REGION

REGION Network 37: Main P&P Job 5 Interface [One Load]
   RUNG wire#powerrail
      Contact( #instMainPnPOneLoadJob5.jobStatus.active )
      Contact( "Unit1.Em5.ControlNodes".cm.softCam.cathodeMainPnP1AxisZ.upPos.inPos )
      Contact( "Unit1.Em5.ControlNodes".cmCathodeMainPnP1SuctionPlateVacuum.monitoring.inWorkPos )
      Coil( "Unit1.Em5.ControlNodes".mainPnP.jobInterface.oneLoadJob5.loadingDone )
   END_RUNG
   RUNG wire#powerrail
      Contact( #instMainPnPOneLoadJob5.jobStatus.active )
      Contact( "Unit1.Em5.ControlNodes".cm.softCam.cathodeMainPnP1AxisZ.reelCutConveyerDownPos.inPos )
      Contact( "Unit1.Em5.ControlNodes".cmCathodeMainPnP1SuctionPlateVacuum.monitoring.inWorkPos )
      Coil( "Unit1.Em5.ControlNodes".mainPnP.jobInterface.oneLoadJob5.loadingReady )
   END_RUNG
   // the same network as SCL:
   "Unit1.Em5.ControlNodes".mainPnP.jobInterface.oneLoadJob5.loadingDone := #instMainPnPOneLoadJob5.jobStatus.active AND "Unit1.Em5.ControlNodes".cm.softCam.cathodeMainPnP1AxisZ.upPos.inPos AND "Unit1.Em5.ControlNodes".cmCathodeMainPnP1SuctionPlateVacuum.monitoring.inWorkPos;
   "Unit1.Em5.ControlNodes".mainPnP.jobInterface.oneLoadJob5.loadingReady := #instMainPnPOneLoadJob5.jobStatus.active AND "Unit1.Em5.ControlNodes".cm.softCam.cathodeMainPnP1AxisZ.reelCutConveyerDownPos.inPos AND "Unit1.Em5.ControlNodes".cmCathodeMainPnP1SuctionPlateVacuum.monitoring.inWorkPos;
END_REGION

REGION Network 38: Main P&P Job 6 Interface [One Unload]
   RUNG wire#powerrail
      I_Contact( #instMainPnPOneUnLoadJob6.jobStatus.active )
      Contact( "Unit1.Em5.ControlNodes".mainPnP."step".action1[650] )
      wire#w1
      Coil( "Unit1.Em5.ControlNodes".mainPnP.jobInterface.oneUnLoadJob6.unLoadingReady )
   END_RUNG
   RUNG wire#powerrail
      Contact( #instMainPnPOneUnLoadJob6.jobStatus.active )
      Contact( "Unit1.Em5.ControlNodes".cm.softCam.cathodeMainPnP1AxisZ.ailgnTableDownPos.inPos )
   END_RUNG wire#w1
   // the same network as SCL:
   "Unit1.Em5.ControlNodes".mainPnP.jobInterface.oneUnLoadJob6.unLoadingReady := (NOT #instMainPnPOneUnLoadJob6.jobStatus.active AND "Unit1.Em5.ControlNodes".mainPnP."step".action1[650]) OR (#instMainPnPOneUnLoadJob6.jobStatus.active AND "Unit1.Em5.ControlNodes".cm.softCam.cathodeMainPnP1AxisZ.ailgnTableDownPos.inPos);
END_REGION

REGION Network 39: Main P&P Job Interface Working Done
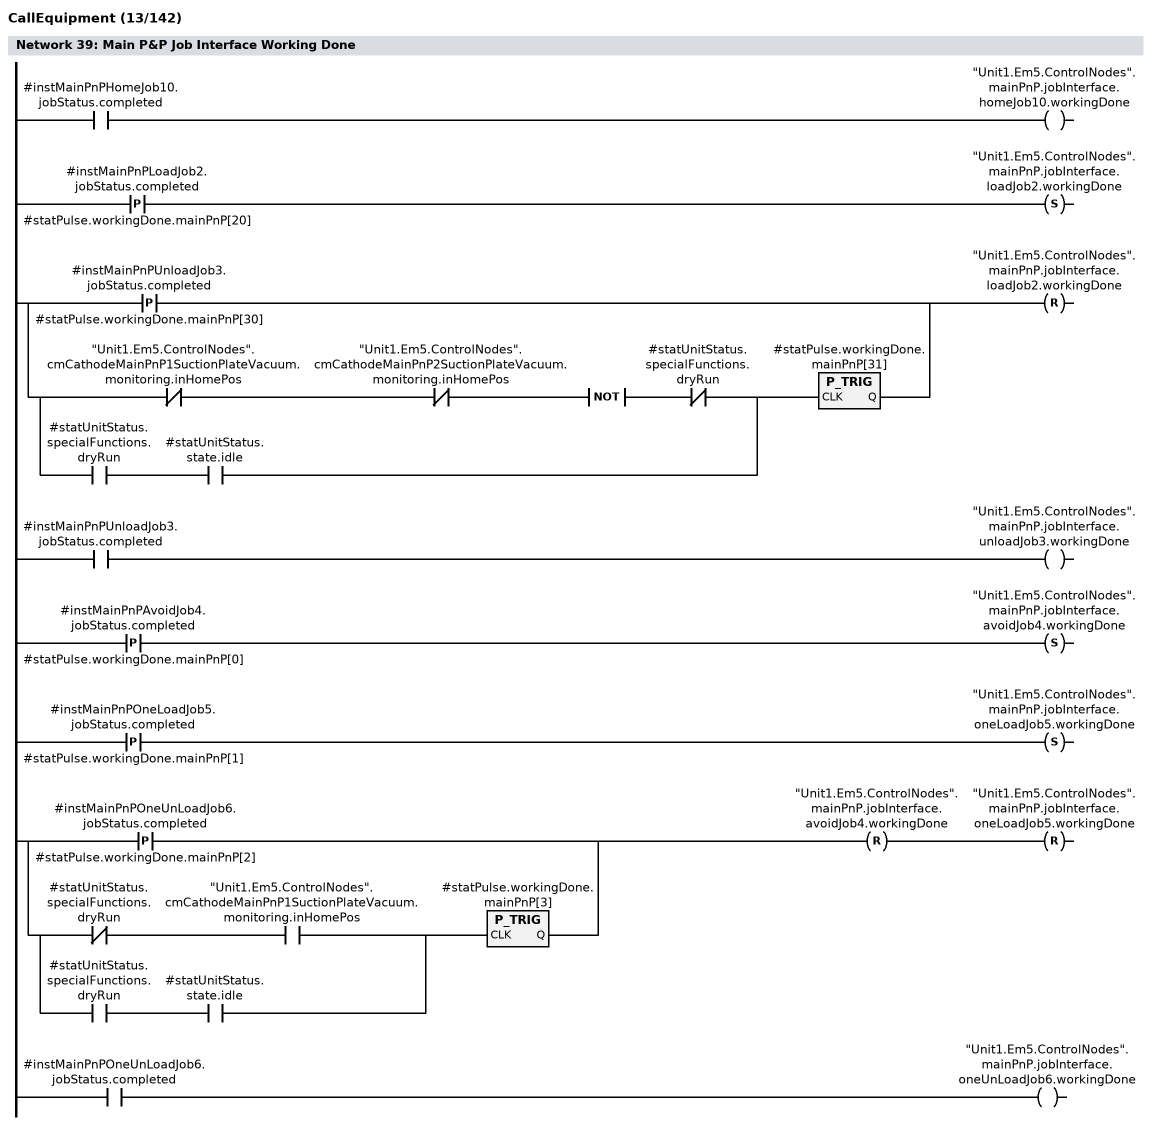
   RUNG wire#powerrail
      Contact( #instMainPnPHomeJob10.jobStatus.completed )
      Coil( "Unit1.Em5.ControlNodes".mainPnP.jobInterface.homeJob10.workingDone )
   END_RUNG
   RUNG wire#powerrail
      P_Contact(operand := #instMainPnPLoadJob2.jobStatus.completed, bit := #statPulse.workingDone.mainPnP[20])
      S_Coil( "Unit1.Em5.ControlNodes".mainPnP.jobInterface.loadJob2.workingDone )
   END_RUNG
   RUNG wire#powerrail
      P_Contact(operand := #instMainPnPUnloadJob3.jobStatus.completed, bit := #statPulse.workingDone.mainPnP[30])
      wire#w1
      R_Coil( "Unit1.Em5.ControlNodes".mainPnP.jobInterface.loadJob2.workingDone )
   END_RUNG
   RUNG wire#powerrail
      I_Contact( "Unit1.Em5.ControlNodes".cmCathodeMainPnP1SuctionPlateVacuum.monitoring.inHomePos )
      I_Contact( "Unit1.Em5.ControlNodes".cmCathodeMainPnP2SuctionPlateVacuum.monitoring.inHomePos )
      Not()
      I_Contact( #statUnitStatus.specialFunctions.dryRun )
      wire#w2
      P_Trig( #statPulse.workingDone.mainPnP[31] )
   END_RUNG wire#w1
   RUNG wire#powerrail
      Contact( #statUnitStatus.specialFunctions.dryRun )
      Contact( #statUnitStatus.state.idle )
   END_RUNG wire#w2
   RUNG wire#powerrail
      Contact( #instMainPnPUnloadJob3.jobStatus.completed )
      Coil( "Unit1.Em5.ControlNodes".mainPnP.jobInterface.unloadJob3.workingDone )
   END_RUNG
   RUNG wire#powerrail
      P_Contact(operand := #instMainPnPAvoidJob4.jobStatus.completed, bit := #statPulse.workingDone.mainPnP[0])
      S_Coil( "Unit1.Em5.ControlNodes".mainPnP.jobInterface.avoidJob4.workingDone )
   END_RUNG
   RUNG wire#powerrail
      P_Contact(operand := #instMainPnPOneLoadJob5.jobStatus.completed, bit := #statPulse.workingDone.mainPnP[1])
      S_Coil( "Unit1.Em5.ControlNodes".mainPnP.jobInterface.oneLoadJob5.workingDone )
   END_RUNG
   RUNG wire#powerrail
      P_Contact(operand := #instMainPnPOneUnLoadJob6.jobStatus.completed, bit := #statPulse.workingDone.mainPnP[2])
      wire#w3
      R_Coil( "Unit1.Em5.ControlNodes".mainPnP.jobInterface.avoidJob4.workingDone )
      R_Coil( "Unit1.Em5.ControlNodes".mainPnP.jobInterface.oneLoadJob5.workingDone )
   END_RUNG
   RUNG wire#powerrail
      I_Contact( #statUnitStatus.specialFunctions.dryRun )
      Contact( "Unit1.Em5.ControlNodes".cmCathodeMainPnP1SuctionPlateVacuum.monitoring.inHomePos )
      wire#w4
      P_Trig( #statPulse.workingDone.mainPnP[3] )
   END_RUNG wire#w3
   RUNG wire#powerrail
      Contact( #statUnitStatus.specialFunctions.dryRun )
      Contact( #statUnitStatus.state.idle )
   END_RUNG wire#w4
   RUNG wire#powerrail
      Contact( #instMainPnPOneUnLoadJob6.jobStatus.completed )
      Coil( "Unit1.Em5.ControlNodes".mainPnP.jobInterface.oneUnLoadJob6.workingDone )
   END_RUNG
   // the same network as SCL:
   "Unit1.Em5.ControlNodes".mainPnP.jobInterface.homeJob10.workingDone := #instMainPnPHomeJob10.jobStatus.completed;
   #_w1 := #instMainPnPLoadJob2.jobStatus.completed AND NOT #statPulse.workingDone.mainPnP[20];   // rising edge of #instMainPnPLoadJob2.jobStatus.completed
   #statPulse.workingDone.mainPnP[20] := #instMainPnPLoadJob2.jobStatus.completed;
   IF #_w1 THEN "Unit1.Em5.ControlNodes".mainPnP.jobInterface.loadJob2.workingDone := TRUE; END_IF;
   #_w2 := #instMainPnPUnloadJob3.jobStatus.completed AND NOT #statPulse.workingDone.mainPnP[30];   // rising edge of #instMainPnPUnloadJob3.jobStatus.completed
   #statPulse.workingDone.mainPnP[30] := #instMainPnPUnloadJob3.jobStatus.completed;
   #_w3 := (NOT (NOT "Unit1.Em5.ControlNodes".cmCathodeMainPnP1SuctionPlateVacuum.monitoring.inHomePos AND NOT "Unit1.Em5.ControlNodes".cmCathodeMainPnP2SuctionPlateVacuum.monitoring.inHomePos) AND NOT #statUnitStatus.specialFunctions.dryRun) OR (#statUnitStatus.specialFunctions.dryRun AND #statUnitStatus.state.idle);
   #_w4 := #_w3 AND NOT #statPulse.workingDone.mainPnP[31];   // rising edge
   #statPulse.workingDone.mainPnP[31] := #_w3;
   IF #_w2 OR #_w4 THEN "Unit1.Em5.ControlNodes".mainPnP.jobInterface.loadJob2.workingDone := FALSE; END_IF;
   "Unit1.Em5.ControlNodes".mainPnP.jobInterface.unloadJob3.workingDone := #instMainPnPUnloadJob3.jobStatus.completed;
   #_w5 := #instMainPnPAvoidJob4.jobStatus.completed AND NOT #statPulse.workingDone.mainPnP[0];   // rising edge of #instMainPnPAvoidJob4.jobStatus.completed
   #statPulse.workingDone.mainPnP[0] := #instMainPnPAvoidJob4.jobStatus.completed;
   IF #_w5 THEN "Unit1.Em5.ControlNodes".mainPnP.jobInterface.avoidJob4.workingDone := TRUE; END_IF;
   #_w6 := #instMainPnPOneLoadJob5.jobStatus.completed AND NOT #statPulse.workingDone.mainPnP[1];   // rising edge of #instMainPnPOneLoadJob5.jobStatus.completed
   #statPulse.workingDone.mainPnP[1] := #instMainPnPOneLoadJob5.jobStatus.completed;
   IF #_w6 THEN "Unit1.Em5.ControlNodes".mainPnP.jobInterface.oneLoadJob5.workingDone := TRUE; END_IF;
   #_w7 := #instMainPnPOneUnLoadJob6.jobStatus.completed AND NOT #statPulse.workingDone.mainPnP[2];   // rising edge of #instMainPnPOneUnLoadJob6.jobStatus.completed
   #statPulse.workingDone.mainPnP[2] := #instMainPnPOneUnLoadJob6.jobStatus.completed;
   #_w8 := (NOT #statUnitStatus.specialFunctions.dryRun AND "Unit1.Em5.ControlNodes".cmCathodeMainPnP1SuctionPlateVacuum.monitoring.inHomePos) OR (#statUnitStatus.specialFunctions.dryRun AND #statUnitStatus.state.idle);
   #_w9 := #_w8 AND NOT #statPulse.workingDone.mainPnP[3];   // rising edge
   #statPulse.workingDone.mainPnP[3] := #_w8;
   IF #_w7 OR #_w9 THEN
       "Unit1.Em5.ControlNodes".mainPnP.jobInterface.avoidJob4.workingDone := FALSE;
       "Unit1.Em5.ControlNodes".mainPnP.jobInterface.oneLoadJob5.workingDone := FALSE;
   END_IF;
   "Unit1.Em5.ControlNodes".mainPnP.jobInterface.oneUnLoadJob6.workingDone := #instMainPnPOneUnLoadJob6.jobStatus.completed;
END_REGION

REGION Network 40: Main P&P Previous Operation Check
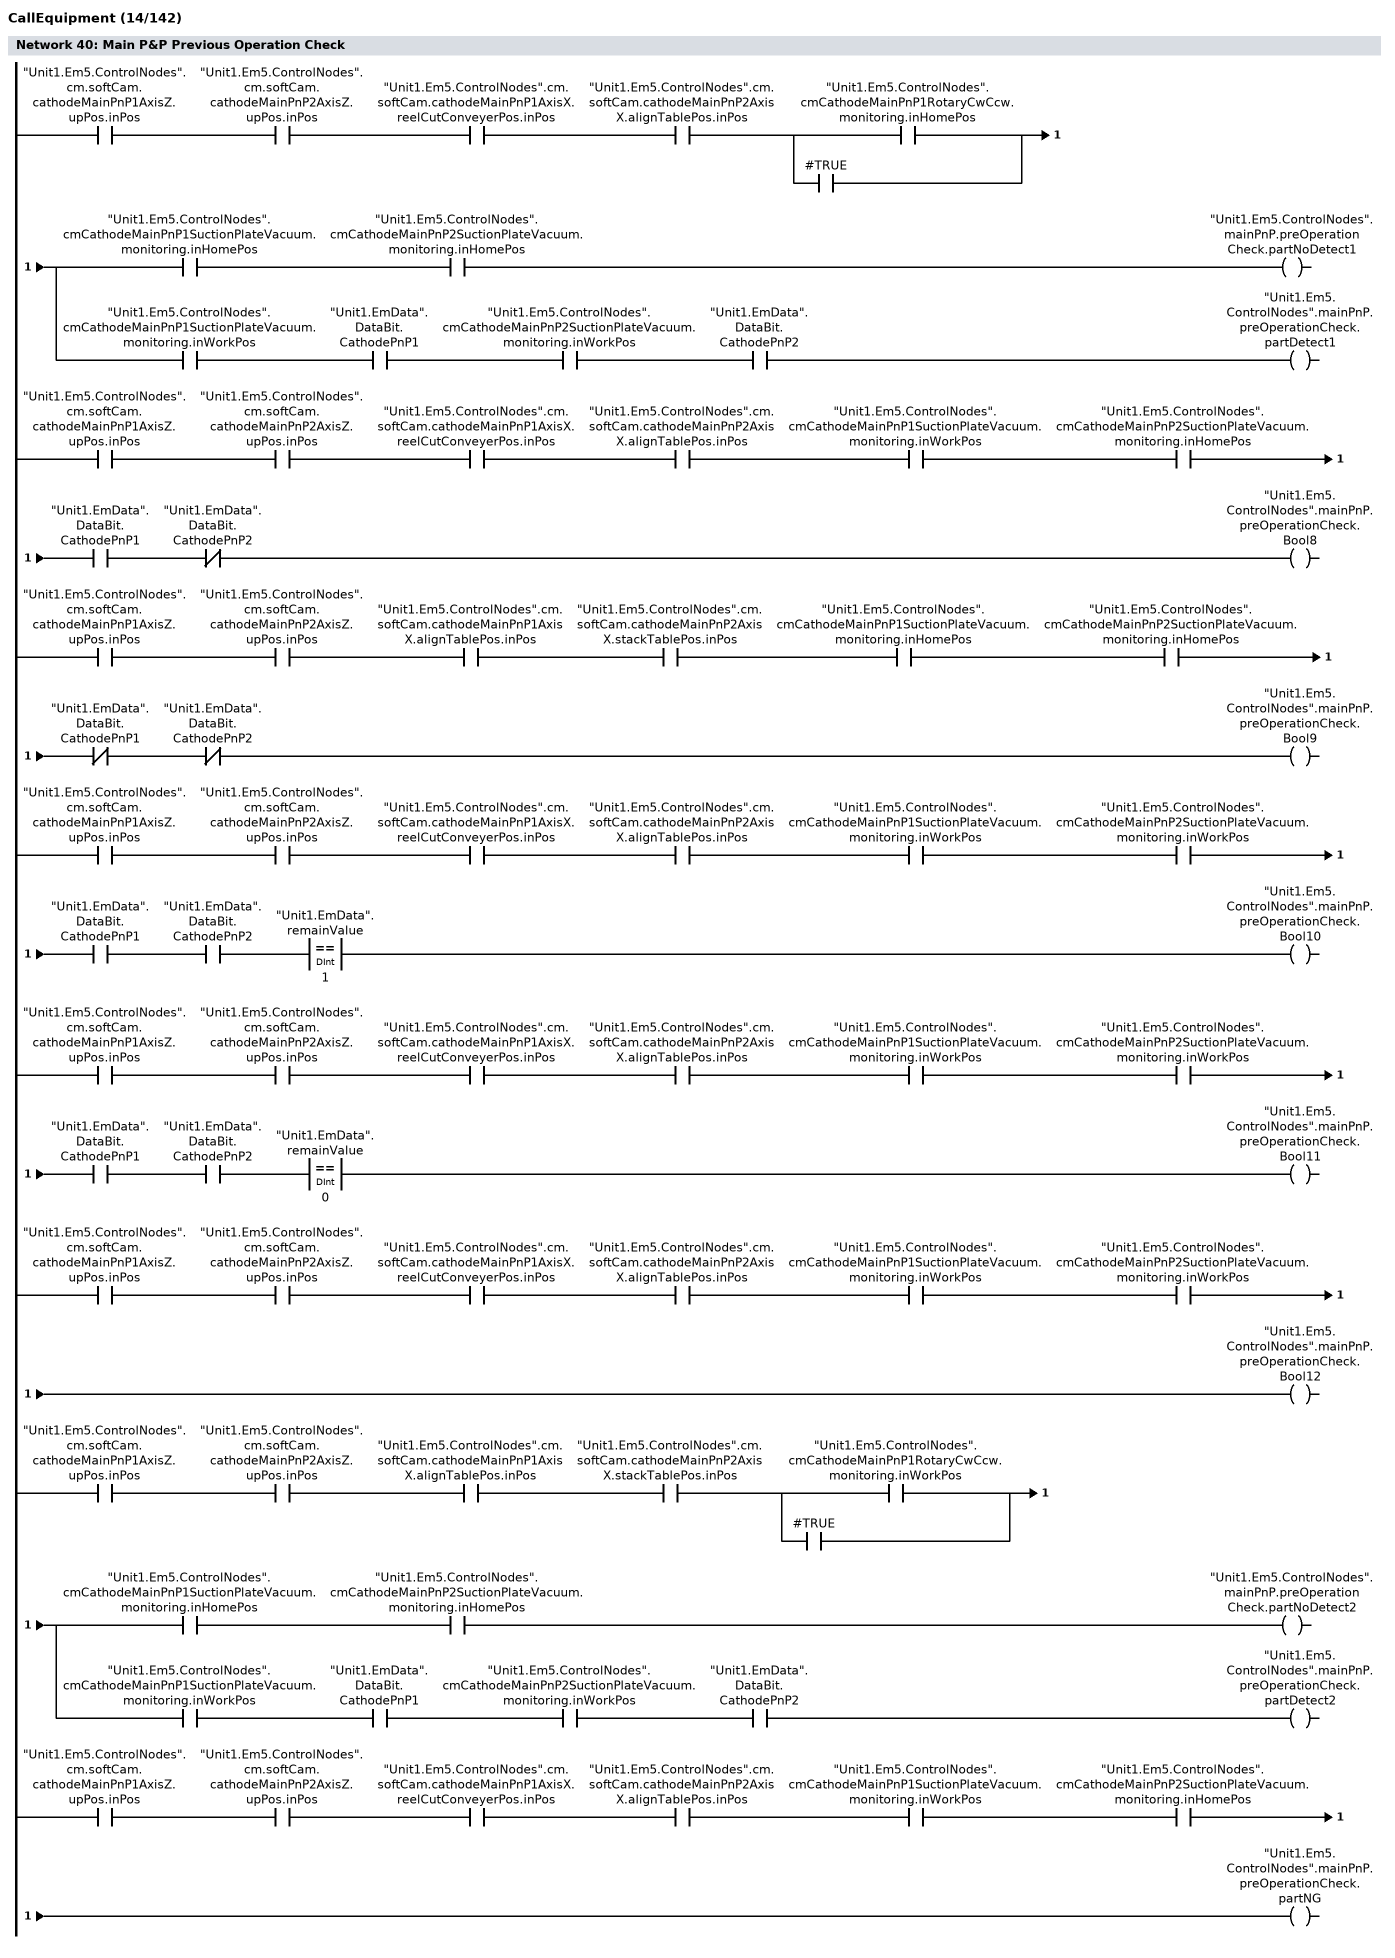
   RUNG wire#powerrail
      Contact( "Unit1.Em5.ControlNodes".cm.softCam.cathodeMainPnP1AxisZ.upPos.inPos )
      Contact( "Unit1.Em5.ControlNodes".cm.softCam.cathodeMainPnP2AxisZ.upPos.inPos )
      Contact( "Unit1.Em5.ControlNodes".cm.softCam.cathodeMainPnP1AxisX.reelCutConveyerPos.inPos )
      Contact( "Unit1.Em5.ControlNodes".cm.softCam.cathodeMainPnP2AxisX.alignTablePos.inPos )
      wire#w1
      Contact( "Unit1.Em5.ControlNodes".cmCathodeMainPnP1RotaryCwCcw.monitoring.inHomePos )
      wire#w2
      Contact( "Unit1.Em5.ControlNodes".cmCathodeMainPnP1SuctionPlateVacuum.monitoring.inHomePos )
      Contact( "Unit1.Em5.ControlNodes".cmCathodeMainPnP2SuctionPlateVacuum.monitoring.inHomePos )
      Coil( "Unit1.Em5.ControlNodes".mainPnP.preOperationCheck.partNoDetect1 )
   END_RUNG
   RUNG wire#w1
      Contact( #TRUE )
   END_RUNG wire#w2
   RUNG wire#w2
      Contact( "Unit1.Em5.ControlNodes".cmCathodeMainPnP1SuctionPlateVacuum.monitoring.inWorkPos )
      Contact( "Unit1.EmData".DataBit.CathodePnP1 )
      Contact( "Unit1.Em5.ControlNodes".cmCathodeMainPnP2SuctionPlateVacuum.monitoring.inWorkPos )
      Contact( "Unit1.EmData".DataBit.CathodePnP2 )
      Coil( "Unit1.Em5.ControlNodes".mainPnP.preOperationCheck.partDetect1 )
   END_RUNG
   RUNG wire#powerrail
      Contact( "Unit1.Em5.ControlNodes".cm.softCam.cathodeMainPnP1AxisZ.upPos.inPos )
      Contact( "Unit1.Em5.ControlNodes".cm.softCam.cathodeMainPnP2AxisZ.upPos.inPos )
      Contact( "Unit1.Em5.ControlNodes".cm.softCam.cathodeMainPnP1AxisX.reelCutConveyerPos.inPos )
      Contact( "Unit1.Em5.ControlNodes".cm.softCam.cathodeMainPnP2AxisX.alignTablePos.inPos )
      Contact( "Unit1.Em5.ControlNodes".cmCathodeMainPnP1SuctionPlateVacuum.monitoring.inWorkPos )
      Contact( "Unit1.Em5.ControlNodes".cmCathodeMainPnP2SuctionPlateVacuum.monitoring.inHomePos )
      Contact( "Unit1.EmData".DataBit.CathodePnP1 )
      I_Contact( "Unit1.EmData".DataBit.CathodePnP2 )
      Coil( "Unit1.Em5.ControlNodes".mainPnP.preOperationCheck.Bool8 )
   END_RUNG
   RUNG wire#powerrail
      Contact( "Unit1.Em5.ControlNodes".cm.softCam.cathodeMainPnP1AxisZ.upPos.inPos )
      Contact( "Unit1.Em5.ControlNodes".cm.softCam.cathodeMainPnP2AxisZ.upPos.inPos )
      Contact( "Unit1.Em5.ControlNodes".cm.softCam.cathodeMainPnP1AxisX.alignTablePos.inPos )
      Contact( "Unit1.Em5.ControlNodes".cm.softCam.cathodeMainPnP2AxisX.stackTablePos.inPos )
      Contact( "Unit1.Em5.ControlNodes".cmCathodeMainPnP1SuctionPlateVacuum.monitoring.inHomePos )
      Contact( "Unit1.Em5.ControlNodes".cmCathodeMainPnP2SuctionPlateVacuum.monitoring.inHomePos )
      I_Contact( "Unit1.EmData".DataBit.CathodePnP1 )
      I_Contact( "Unit1.EmData".DataBit.CathodePnP2 )
      Coil( "Unit1.Em5.ControlNodes".mainPnP.preOperationCheck.Bool9 )
   END_RUNG
   RUNG wire#powerrail
      Contact( "Unit1.Em5.ControlNodes".cm.softCam.cathodeMainPnP1AxisZ.upPos.inPos )
      Contact( "Unit1.Em5.ControlNodes".cm.softCam.cathodeMainPnP2AxisZ.upPos.inPos )
      Contact( "Unit1.Em5.ControlNodes".cm.softCam.cathodeMainPnP1AxisX.reelCutConveyerPos.inPos )
      Contact( "Unit1.Em5.ControlNodes".cm.softCam.cathodeMainPnP2AxisX.alignTablePos.inPos )
      Contact( "Unit1.Em5.ControlNodes".cmCathodeMainPnP1SuctionPlateVacuum.monitoring.inWorkPos )
      Contact( "Unit1.Em5.ControlNodes".cmCathodeMainPnP2SuctionPlateVacuum.monitoring.inWorkPos )
      Contact( "Unit1.EmData".DataBit.CathodePnP1 )
      Contact( "Unit1.EmData".DataBit.CathodePnP2 )
      { S7_Templates := "SrcType := DInt" } EQ_Contact(in1 := "Unit1.EmData".remainValue, in2 := 1)
      Coil( "Unit1.Em5.ControlNodes".mainPnP.preOperationCheck.Bool10 )
   END_RUNG
   RUNG wire#powerrail
      Contact( "Unit1.Em5.ControlNodes".cm.softCam.cathodeMainPnP1AxisZ.upPos.inPos )
      Contact( "Unit1.Em5.ControlNodes".cm.softCam.cathodeMainPnP2AxisZ.upPos.inPos )
      Contact( "Unit1.Em5.ControlNodes".cm.softCam.cathodeMainPnP1AxisX.reelCutConveyerPos.inPos )
      Contact( "Unit1.Em5.ControlNodes".cm.softCam.cathodeMainPnP2AxisX.alignTablePos.inPos )
      Contact( "Unit1.Em5.ControlNodes".cmCathodeMainPnP1SuctionPlateVacuum.monitoring.inWorkPos )
      Contact( "Unit1.Em5.ControlNodes".cmCathodeMainPnP2SuctionPlateVacuum.monitoring.inWorkPos )
      Contact( "Unit1.EmData".DataBit.CathodePnP1 )
      Contact( "Unit1.EmData".DataBit.CathodePnP2 )
      { S7_Templates := "SrcType := DInt" } EQ_Contact(in1 := "Unit1.EmData".remainValue, in2 := 0)
      Coil( "Unit1.Em5.ControlNodes".mainPnP.preOperationCheck.Bool11 )
   END_RUNG
   RUNG wire#powerrail
      Contact( "Unit1.Em5.ControlNodes".cm.softCam.cathodeMainPnP1AxisZ.upPos.inPos )
      Contact( "Unit1.Em5.ControlNodes".cm.softCam.cathodeMainPnP2AxisZ.upPos.inPos )
      Contact( "Unit1.Em5.ControlNodes".cm.softCam.cathodeMainPnP1AxisX.reelCutConveyerPos.inPos )
      Contact( "Unit1.Em5.ControlNodes".cm.softCam.cathodeMainPnP2AxisX.alignTablePos.inPos )
      Contact( "Unit1.Em5.ControlNodes".cmCathodeMainPnP1SuctionPlateVacuum.monitoring.inWorkPos )
      Contact( "Unit1.Em5.ControlNodes".cmCathodeMainPnP2SuctionPlateVacuum.monitoring.inWorkPos )
      Coil( "Unit1.Em5.ControlNodes".mainPnP.preOperationCheck.Bool12 )
   END_RUNG
   RUNG wire#powerrail
      Contact( "Unit1.Em5.ControlNodes".cm.softCam.cathodeMainPnP1AxisZ.upPos.inPos )
      Contact( "Unit1.Em5.ControlNodes".cm.softCam.cathodeMainPnP2AxisZ.upPos.inPos )
      Contact( "Unit1.Em5.ControlNodes".cm.softCam.cathodeMainPnP1AxisX.alignTablePos.inPos )
      Contact( "Unit1.Em5.ControlNodes".cm.softCam.cathodeMainPnP2AxisX.stackTablePos.inPos )
      wire#w3
      Contact( "Unit1.Em5.ControlNodes".cmCathodeMainPnP1RotaryCwCcw.monitoring.inWorkPos )
      wire#w4
      Contact( "Unit1.Em5.ControlNodes".cmCathodeMainPnP1SuctionPlateVacuum.monitoring.inHomePos )
      Contact( "Unit1.Em5.ControlNodes".cmCathodeMainPnP2SuctionPlateVacuum.monitoring.inHomePos )
      Coil( "Unit1.Em5.ControlNodes".mainPnP.preOperationCheck.partNoDetect2 )
   END_RUNG
   RUNG wire#w3
      Contact( #TRUE )
   END_RUNG wire#w4
   RUNG wire#w4
      Contact( "Unit1.Em5.ControlNodes".cmCathodeMainPnP1SuctionPlateVacuum.monitoring.inWorkPos )
      Contact( "Unit1.EmData".DataBit.CathodePnP1 )
      Contact( "Unit1.Em5.ControlNodes".cmCathodeMainPnP2SuctionPlateVacuum.monitoring.inWorkPos )
      Contact( "Unit1.EmData".DataBit.CathodePnP2 )
      Coil( "Unit1.Em5.ControlNodes".mainPnP.preOperationCheck.partDetect2 )
   END_RUNG
   RUNG wire#powerrail
      Contact( "Unit1.Em5.ControlNodes".cm.softCam.cathodeMainPnP1AxisZ.upPos.inPos )
      Contact( "Unit1.Em5.ControlNodes".cm.softCam.cathodeMainPnP2AxisZ.upPos.inPos )
      Contact( "Unit1.Em5.ControlNodes".cm.softCam.cathodeMainPnP1AxisX.reelCutConveyerPos.inPos )
      Contact( "Unit1.Em5.ControlNodes".cm.softCam.cathodeMainPnP2AxisX.alignTablePos.inPos )
      Contact( "Unit1.Em5.ControlNodes".cmCathodeMainPnP1SuctionPlateVacuum.monitoring.inWorkPos )
      Contact( "Unit1.Em5.ControlNodes".cmCathodeMainPnP2SuctionPlateVacuum.monitoring.inHomePos )
      Coil( "Unit1.Em5.ControlNodes".mainPnP.preOperationCheck.partNG )
   END_RUNG
   // the same network as SCL:
   #_w1 := "Unit1.Em5.ControlNodes".cm.softCam.cathodeMainPnP1AxisZ.upPos.inPos AND "Unit1.Em5.ControlNodes".cm.softCam.cathodeMainPnP2AxisZ.upPos.inPos AND "Unit1.Em5.ControlNodes".cm.softCam.cathodeMainPnP1AxisX.reelCutConveyerPos.inPos AND "Unit1.Em5.ControlNodes".cm.softCam.cathodeMainPnP2AxisX.alignTablePos.inPos AND ("Unit1.Em5.ControlNodes".cmCathodeMainPnP1RotaryCwCcw.monitoring.inHomePos OR #TRUE);
   "Unit1.Em5.ControlNodes".mainPnP.preOperationCheck.partNoDetect1 := #_w1 AND "Unit1.Em5.ControlNodes".cmCathodeMainPnP1SuctionPlateVacuum.monitoring.inHomePos AND "Unit1.Em5.ControlNodes".cmCathodeMainPnP2SuctionPlateVacuum.monitoring.inHomePos;
   "Unit1.Em5.ControlNodes".mainPnP.preOperationCheck.partDetect1 := #_w1 AND "Unit1.Em5.ControlNodes".cmCathodeMainPnP1SuctionPlateVacuum.monitoring.inWorkPos AND "Unit1.EmData".DataBit.CathodePnP1 AND "Unit1.Em5.ControlNodes".cmCathodeMainPnP2SuctionPlateVacuum.monitoring.inWorkPos AND "Unit1.EmData".DataBit.CathodePnP2;
   "Unit1.Em5.ControlNodes".mainPnP.preOperationCheck.Bool8 := "Unit1.Em5.ControlNodes".cm.softCam.cathodeMainPnP1AxisZ.upPos.inPos AND "Unit1.Em5.ControlNodes".cm.softCam.cathodeMainPnP2AxisZ.upPos.inPos AND "Unit1.Em5.ControlNodes".cm.softCam.cathodeMainPnP1AxisX.reelCutConveyerPos.inPos AND "Unit1.Em5.ControlNodes".cm.softCam.cathodeMainPnP2AxisX.alignTablePos.inPos AND "Unit1.Em5.ControlNodes".cmCathodeMainPnP1SuctionPlateVacuum.monitoring.inWorkPos AND "Unit1.Em5.ControlNodes".cmCathodeMainPnP2SuctionPlateVacuum.monitoring.inHomePos AND "Unit1.EmData".DataBit.CathodePnP1 AND NOT "Unit1.EmData".DataBit.CathodePnP2;
   "Unit1.Em5.ControlNodes".mainPnP.preOperationCheck.Bool9 := "Unit1.Em5.ControlNodes".cm.softCam.cathodeMainPnP1AxisZ.upPos.inPos AND "Unit1.Em5.ControlNodes".cm.softCam.cathodeMainPnP2AxisZ.upPos.inPos AND "Unit1.Em5.ControlNodes".cm.softCam.cathodeMainPnP1AxisX.alignTablePos.inPos AND "Unit1.Em5.ControlNodes".cm.softCam.cathodeMainPnP2AxisX.stackTablePos.inPos AND "Unit1.Em5.ControlNodes".cmCathodeMainPnP1SuctionPlateVacuum.monitoring.inHomePos AND "Unit1.Em5.ControlNodes".cmCathodeMainPnP2SuctionPlateVacuum.monitoring.inHomePos AND NOT "Unit1.EmData".DataBit.CathodePnP1 AND NOT "Unit1.EmData".DataBit.CathodePnP2;
   "Unit1.Em5.ControlNodes".mainPnP.preOperationCheck.Bool10 := "Unit1.Em5.ControlNodes".cm.softCam.cathodeMainPnP1AxisZ.upPos.inPos AND "Unit1.Em5.ControlNodes".cm.softCam.cathodeMainPnP2AxisZ.upPos.inPos AND "Unit1.Em5.ControlNodes".cm.softCam.cathodeMainPnP1AxisX.reelCutConveyerPos.inPos AND "Unit1.Em5.ControlNodes".cm.softCam.cathodeMainPnP2AxisX.alignTablePos.inPos AND "Unit1.Em5.ControlNodes".cmCathodeMainPnP1SuctionPlateVacuum.monitoring.inWorkPos AND "Unit1.Em5.ControlNodes".cmCathodeMainPnP2SuctionPlateVacuum.monitoring.inWorkPos AND "Unit1.EmData".DataBit.CathodePnP1 AND "Unit1.EmData".DataBit.CathodePnP2 AND ("Unit1.EmData".remainValue = 1);
   "Unit1.Em5.ControlNodes".mainPnP.preOperationCheck.Bool11 := "Unit1.Em5.ControlNodes".cm.softCam.cathodeMainPnP1AxisZ.upPos.inPos AND "Unit1.Em5.ControlNodes".cm.softCam.cathodeMainPnP2AxisZ.upPos.inPos AND "Unit1.Em5.ControlNodes".cm.softCam.cathodeMainPnP1AxisX.reelCutConveyerPos.inPos AND "Unit1.Em5.ControlNodes".cm.softCam.cathodeMainPnP2AxisX.alignTablePos.inPos AND "Unit1.Em5.ControlNodes".cmCathodeMainPnP1SuctionPlateVacuum.monitoring.inWorkPos AND "Unit1.Em5.ControlNodes".cmCathodeMainPnP2SuctionPlateVacuum.monitoring.inWorkPos AND "Unit1.EmData".DataBit.CathodePnP1 AND "Unit1.EmData".DataBit.CathodePnP2 AND ("Unit1.EmData".remainValue = 0);
   "Unit1.Em5.ControlNodes".mainPnP.preOperationCheck.Bool12 := "Unit1.Em5.ControlNodes".cm.softCam.cathodeMainPnP1AxisZ.upPos.inPos AND "Unit1.Em5.ControlNodes".cm.softCam.cathodeMainPnP2AxisZ.upPos.inPos AND "Unit1.Em5.ControlNodes".cm.softCam.cathodeMainPnP1AxisX.reelCutConveyerPos.inPos AND "Unit1.Em5.ControlNodes".cm.softCam.cathodeMainPnP2AxisX.alignTablePos.inPos AND "Unit1.Em5.ControlNodes".cmCathodeMainPnP1SuctionPlateVacuum.monitoring.inWorkPos AND "Unit1.Em5.ControlNodes".cmCathodeMainPnP2SuctionPlateVacuum.monitoring.inWorkPos;
   #_w2 := "Unit1.Em5.ControlNodes".cm.softCam.cathodeMainPnP1AxisZ.upPos.inPos AND "Unit1.Em5.ControlNodes".cm.softCam.cathodeMainPnP2AxisZ.upPos.inPos AND "Unit1.Em5.ControlNodes".cm.softCam.cathodeMainPnP1AxisX.alignTablePos.inPos AND "Unit1.Em5.ControlNodes".cm.softCam.cathodeMainPnP2AxisX.stackTablePos.inPos AND ("Unit1.Em5.ControlNodes".cmCathodeMainPnP1RotaryCwCcw.monitoring.inWorkPos OR #TRUE);
   "Unit1.Em5.ControlNodes".mainPnP.preOperationCheck.partNoDetect2 := #_w2 AND "Unit1.Em5.ControlNodes".cmCathodeMainPnP1SuctionPlateVacuum.monitoring.inHomePos AND "Unit1.Em5.ControlNodes".cmCathodeMainPnP2SuctionPlateVacuum.monitoring.inHomePos;
   "Unit1.Em5.ControlNodes".mainPnP.preOperationCheck.partDetect2 := #_w2 AND "Unit1.Em5.ControlNodes".cmCathodeMainPnP1SuctionPlateVacuum.monitoring.inWorkPos AND "Unit1.EmData".DataBit.CathodePnP1 AND "Unit1.Em5.ControlNodes".cmCathodeMainPnP2SuctionPlateVacuum.monitoring.inWorkPos AND "Unit1.EmData".DataBit.CathodePnP2;
   "Unit1.Em5.ControlNodes".mainPnP.preOperationCheck.partNG := "Unit1.Em5.ControlNodes".cm.softCam.cathodeMainPnP1AxisZ.upPos.inPos AND "Unit1.Em5.ControlNodes".cm.softCam.cathodeMainPnP2AxisZ.upPos.inPos AND "Unit1.Em5.ControlNodes".cm.softCam.cathodeMainPnP1AxisX.reelCutConveyerPos.inPos AND "Unit1.Em5.ControlNodes".cm.softCam.cathodeMainPnP2AxisX.alignTablePos.inPos AND "Unit1.Em5.ControlNodes".cmCathodeMainPnP1SuctionPlateVacuum.monitoring.inWorkPos AND "Unit1.Em5.ControlNodes".cmCathodeMainPnP2SuctionPlateVacuum.monitoring.inHomePos;
END_REGION

